LIN {X 0,Y 504.63,Z 384.162,A -85,B 0,C 180,E1 24334.794,E2 24334.794} C_VEL
LIN {X 0,Y 504.69,Z 384.156,A -85,B 0,C 180,E1 24331.534,E2 24331.534} C_VEL
LIN {X 0,Y 504.631,Z 384.188,A -85,B 0,C 180,E1 24328.264,E2 24328.264} C_VEL
LIN {X 0,Y 504.665,Z 384.158,A -85,B 0,C 180,E1 24324.835,E2 24324.835} C_VEL
LIN {X 0,Y 504.642,Z 384.183,A -85,B 0,C 180,E1 24321.624,E2 24321.624} C_VEL
LIN {X 0,Y 504.635,Z 384.173,A -85,B 0,C 180,E1 24318.123,E2 24318.123} C_VEL
LIN {X 0,Y 504.698,Z 384.163,A -85,B 0,C 180,E1 24314.806,E2 24314.806} C_VEL
LIN {X 0,Y 504.631,Z 384.169,A -85,B 0,C 180,E1 24311.428,E2 24311.428} C_VEL
LIN {X 0,Y 504.655,Z 384.173,A -85,B 0,C 180,E1 24307.972,E2 24307.972} C_VEL
LIN {X 0,Y 504.654,Z 384.182,A -85,B 0,C 180,E1 24304.773,E2 24304.773} C_VEL
LIN {X 0,Y 504.638,Z 384.181,A -85,B 0,C 180,E1 24301.362,E2 24301.362} C_VEL
LIN {X 0,Y 504.698,Z 384.182,A -85,B 0,C 180,E1 24298.07,E2 24298.07} C_VEL
LIN {X 0,Y 504.638,Z 384.185,A -85,B 0,C 180,E1 24294.656,E2 24294.656} C_VEL
LIN {X 0,Y 504.65,Z 384.184,A -85,B 0,C 180,E1 24291.11,E2 24291.11} C_VEL
LIN {X 0,Y 504.686,Z 384.178,A -85,B 0,C 180,E1 24287.761,E2 24287.761} C_VEL
LIN {X 0,Y 504.637,Z 384.18,A -85,B 0,C 180,E1 24284.485,E2 24284.485} C_VEL
LIN {X 0,Y 504.698,Z 384.175,A -85,B 0,C 180,E1 24281.16,E2 24281.16} C_VEL
LIN {X 0,Y 504.641,Z 384.178,A -85,B 0,C 180,E1 24277.886,E2 24277.886} C_VEL
LIN {X 0,Y 504.651,Z 384.179,A -85,B 0,C 180,E1 24274.355,E2 24274.355} C_VEL
LIN {X 0,Y 504.681,Z 384.161,A -85,B 0,C 180,E1 24271.092,E2 24271.092} C_VEL
LIN {X 0,Y 504.641,Z 384.182,A -85,B 0,C 180,E1 24267.659,E2 24267.659} C_VEL
LIN {X 0,Y 504.678,Z 384.151,A -85,B 0,C 180,E1 24264.236,E2 24264.236} C_VEL
LIN {X 0,Y 504.657,Z 384.186,A -85,B 0,C 180,E1 24260.946,E2 24260.946} C_VEL
LIN {X 0,Y 504.647,Z 384.176,A -85,B 0,C 180,E1 24257.481,E2 24257.481} C_VEL
LIN {X 0,Y 504.699,Z 384.152,A -85,B 0,C 180,E1 24254.148,E2 24254.148} C_VEL
LIN {X 0,Y 504.712,Z 384.421,A -85,B 0,C 180,E1 24252.343,E2 24252.343} C_VEL
LIN {X 0,Y 505.96,Z 387.581,A -85,B 0,C 180,E1 24251.839,E2 24251.839} C_VEL
LIN {X 0,Y 506.781,Z 388.94,A -85,B 0,C 180,E1 24251.616,E2 24251.616} C_VEL
LIN {X 0,Y 508.029,Z 395.982,A -85,B 0,C 180,E1 24250.823,E2 24250.823} C_VEL
LIN {X 0,Y 509.186,Z 410.16,A -85,B 0,C 180,E1 24249.409,E2 24249.409} C_VEL
LIN {X 0,Y 510.462,Z 414.617,A -85,B 0,C 180,E1 24248.871,E2 24248.871} C_VEL
LIN {X 0,Y 513.393,Z 421.793,A -85,B 0,C 180,E1 24247.93,E2 24247.93} C_VEL
LIN {X 0,Y 510.149,Z 468.492,A -85,B 0,C 180,E1 24244.297,E2 24244.297} C_VEL
LIN {X 0,Y 510.416,Z 471.577,A -85,B 0,C 180,E1 24244.143,E2 24244.143} C_VEL
LIN {X 0,Y 513.342,Z 489.328,A -85,B 0,C 180,E1 24243.576,E2 24243.576} C_VEL
LIN {X 0,Y 510.537,Z 702.166,A -85,B 0,C 180,E1 24240.34,E2 24240.34} C_VEL
LIN {X 0,Y 509.946,Z 737.203,A -85,B 0,C 180,E1 24239.76,E2 24239.76} C_VEL
LIN {X 0,Y 509.167,Z 757.239,A -85,B 0,C 180,E1 24239.22,E2 24239.22} C_VEL
LIN {X 0,Y 508.146,Z 775.437,A -85,B 0,C 180,E1 24238.532,E2 24238.532} C_VEL
LIN {X 0,Y 506.819,Z 794.151,A -85,B 0,C 180,E1 24237.621,E2 24237.621} C_VEL
LIN {X 0,Y 505.413,Z 811.582,A -85,B 0,C 180,E1 24236.558,E2 24236.558} C_VEL
LIN {X 0,Y 503.7,Z 829.704,A -85,B 0,C 180,E1 24235.201,E2 24235.201} C_VEL
LIN {X 0,Y 502.073,Z 846.017,A -85,B 0,C 180,E1 24233.721,E2 24233.721} C_VEL
LIN {X 0,Y 500.46,Z 861.756,A -85,B 0,C 180,E1 24232.025,E2 24232.025} C_VEL
LIN {X 0,Y 498.795,Z 880.019,A -85,B 0,C 180,E1 24229.68,E2 24229.68} C_VEL
LIN {X 0,Y 497.903,Z 893.059,A -85,B 0,C 180,E1 24227.773,E2 24227.773} C_VEL
LIN {X 0,Y 497.196,Z 904.769,A -85,B 0,C 180,E1 24225.753,E2 24225.753} C_VEL
LIN {X 0,Y 496.636,Z 915.718,A -85,B 0,C 180,E1 24223.49,E2 24223.49} C_VEL
LIN {X 0,Y 496.275,Z 924.505,A -85,B 0,C 180,E1 24221.27,E2 24221.27} C_VEL
LIN {X 0,Y 496.064,Z 931.644,A -85,B 0,C 180,E1 24219.018,E2 24219.018} C_VEL
LIN {X 0,Y 495.966,Z 937.163,A -85,B 0,C 180,E1 24216.715,E2 24216.715} C_VEL
LIN {X 0,Y 495.923,Z 941.025,A -85,B 0,C 180,E1 24214.394,E2 24214.394} C_VEL
LIN {X 0,Y 495.913,Z 943.345,A -85,B 0,C 180,E1 24211.964,E2 24211.964} C_VEL
LIN {X 0,Y 495.903,Z 943.948,A -85,B 0,C 180,E1 24209.653,E2 24209.653} C_VEL
LIN {X 0,Y 495.907,Z 942.989,A -85,B 0,C 180,E1 24207.342,E2 24207.342} C_VEL
LIN {X 0,Y 495.924,Z 940.351,A -85,B 0,C 180,E1 24205.026,E2 24205.026} C_VEL
LIN {X 0,Y 495.968,Z 936.05,A -85,B 0,C 180,E1 24202.686,E2 24202.686} C_VEL
LIN {X 0,Y 496.099,Z 930.109,A -85,B 0,C 180,E1 24200.37,E2 24200.37} C_VEL
LIN {X 0,Y 496.343,Z 922.728,A -85,B 0,C 180,E1 24198.143,E2 24198.143} C_VEL
LIN {X 0,Y 496.74,Z 913.462,A -85,B 0,C 180,E1 24195.904,E2 24195.904} C_VEL
LIN {X 0,Y 497.314,Z 902.703,A -85,B 0,C 180,E1 24193.772,E2 24193.772} C_VEL
LIN {X 0,Y 498.082,Z 890.332,A -85,B 0,C 180,E1 24191.716,E2 24191.716} C_VEL
LIN {X 0,Y 499.412,Z 872.531,A -85,B 0,C 180,E1 24189.224,E2 24189.224} C_VEL
LIN {X 0,Y 500.948,Z 857.086,A -85,B 0,C 180,E1 24187.343,E2 24187.343} C_VEL
LIN {X 0,Y 502.625,Z 840.515,A -85,B 0,C 180,E1 24185.657,E2 24185.657} C_VEL
LIN {X 0,Y 504.236,Z 824.047,A -85,B 0,C 180,E1 24184.262,E2 24184.262} C_VEL
LIN {X 0,Y 505.82,Z 806.472,A -85,B 0,C 180,E1 24183.021,E2 24183.021} C_VEL
LIN {X 0,Y 507.308,Z 787.941,A -85,B 0,C 180,E1 24181.961,E2 24181.961} C_VEL
LIN {X 0,Y 508.538,Z 769.216,A -85,B 0,C 180,E1 24181.114,E2 24181.114} C_VEL
LIN {X 0,Y 509.525,Z 749.435,A -85,B 0,C 180,E1 24180.455,E2 24180.455} C_VEL
LIN {X 0,Y 510.109,Z 729.43,A -85,B 0,C 180,E1 24179.999,E2 24179.999} C_VEL
LIN {X 0,Y 512.344,Z 567.172,A -85,B 0,C 180,E1 24177.509,E2 24177.509} C_VEL
LIN {X 0,Y 513.183,Z 487.495,A -85,B 0,C 180,E1 24176.288,E2 24176.288} C_VEL
LIN {X 0,Y 510.105,Z 469.195,A -85,B 0,C 180,E1 24175.665,E2 24175.665} C_VEL
LIN {X 0,Y 513.299,Z 423.111,A -85,B 0,C 180,E1 24172.083,E2 24172.083} C_VEL
LIN {X 0,Y 513.288,Z 421.061,A -85,B 0,C 180,E1 24171.904,E2 24171.904} C_VEL
LIN {X 0,Y 506.083,Z 405.037,A -85,B 0,C 180,E1 24169.695,E2 24169.695} C_VEL
LIN {X 0,Y 499.801,Z 392.121,A -85,B 0,C 180,E1 24167.748,E2 24167.748} C_VEL
LIN {X 0,Y 498.273,Z 389.006,A -85,B 0,C 180,E1 24167.26,E2 24167.26} C_VEL
LIN {X 0,Y 496.757,Z 385.456,A -85,B 0,C 180,E1 24166.679,E2 24166.679} C_VEL
LIN {X 0,Y 496.718,Z 385.143,A -85,B 0,C 180,E1 24165.208,E2 24165.208} C_VEL
LIN {X 0,Y 496.764,Z 385.142,A -85,B 0,C 180,E1 24161.776,E2 24161.776} C_VEL
LIN {X 0,Y 496.711,Z 385.175,A -85,B 0,C 180,E1 24158.46,E2 24158.46} C_VEL
LIN {X 0,Y 496.732,Z 385.147,A -85,B 0,C 180,E1 24154.991,E2 24154.991} C_VEL
LIN {X 0,Y 496.738,Z 385.152,A -85,B 0,C 180,E1 24151.631,E2 24151.631} C_VEL
LIN {X 0,Y 496.708,Z 385.17,A -85,B 0,C 180,E1 24148.153,E2 24148.153} C_VEL
LIN {X 0,Y 496.752,Z 385.166,A -85,B 0,C 180,E1 24144.75,E2 24144.75} C_VEL
LIN {X 0,Y 496.721,Z 385.165,A -85,B 0,C 180,E1 24141.367,E2 24141.367} C_VEL
LIN {X 0,Y 496.705,Z 385.172,A -85,B 0,C 180,E1 24137.817,E2 24137.817} C_VEL
LIN {X 0,Y 496.769,Z 385.161,A -85,B 0,C 180,E1 24134.453,E2 24134.453} C_VEL
LIN {X 0,Y 496.711,Z 385.162,A -85,B 0,C 180,E1 24131.025,E2 24131.025} C_VEL
LIN {X 0,Y 496.706,Z 385.164,A -85,B 0,C 180,E1 24127.519,E2 24127.519} C_VEL
LIN {X 0,Y 496.76,Z 385.164,A -85,B 0,C 180,E1 24124.156,E2 24124.156} C_VEL
LIN {X 0,Y 496.7,Z 385.172,A -85,B 0,C 180,E1 24120.808,E2 24120.808} C_VEL
LIN {X 0,Y 496.723,Z 385.171,A -85,B 0,C 180,E1 24117.347,E2 24117.347} C_VEL
LIN {X 0,Y 496.732,Z 385.172,A -85,B 0,C 180,E1 24113.992,E2 24113.992} C_VEL
LIN {X 0,Y 496.697,Z 385.174,A -85,B 0,C 180,E1 24110.535,E2 24110.535} C_VEL
LIN {X 0,Y 496.737,Z 385.132,A -85,B 0,C 180,E1 24107.09,E2 24107.09} C_VEL
LIN {X 0,Y 496.704,Z 385.172,A -85,B 0,C 180,E1 24103.872,E2 24103.872} C_VEL
LIN {X 0,Y 496.698,Z 385.138,A -85,B 0,C 180,E1 24100.357,E2 24100.357} C_VEL
LIN {X 0,Y 496.758,Z 385.17,A -85,B 0,C 180,E1 24097.016,E2 24097.016} C_VEL
LIN {X 0,Y 496.693,Z 385.151,A -85,B 0,C 180,E1 24093.585,E2 24093.585} C_VEL
LIN {X 0,Y 496.704,Z 385.148,A -85,B 0,C 180,E1 24090.052,E2 24090.052} C_VEL
LIN {X 0,Y 496.728,Z 385.177,A -85,B 0,C 180,E1 24086.804,E2 24086.804} C_VEL
LIN {X 0,Y 496.689,Z 385.16,A -85,B 0,C 180,E1 24083.426,E2 24083.426} C_VEL
LIN {X 0,Y 496.775,Z 385.4,A -85,B 0,C 180,E1 24082.468,E2 24082.468} C_VEL
LIN {X 0,Y 497.335,Z 387.314,A -85,B 0,C 180,E1 24082.181,E2 24082.181} C_VEL
LIN {X 0,Y 499.538,Z 390.989,A -85,B 0,C 180,E1 24081.649,E2 24081.649} C_VEL
LIN {X 0,Y 507.023,Z 404.592,A -85,B 0,C 180,E1 24079.846,E2 24079.846} C_VEL
LIN {X 0,Y 517.059,Z 423.783,A -85,B 0,C 180,E1 24077.556,E2 24077.556} C_VEL
LIN {X 0,Y 519.732,Z 428.932,A -85,B 0,C 180,E1 24076.974,E2 24076.974} C_VEL
LIN {X 0,Y 518.222,Z 466.463,A -85,B 0,C 180,E1 24074.906,E2 24074.906} C_VEL
LIN {X 0,Y 520.792,Z 487.007,A -85,B 0,C 180,E1 24074.305,E2 24074.305} C_VEL
LIN {X 0,Y 518.435,Z 664.252,A -85,B 0,C 180,E1 24071.478,E2 24071.478} C_VEL
LIN {X 0,Y 516.725,Z 807.877,A -85,B 0,C 180,E1 24069.261,E2 24069.261} C_VEL
LIN {X 0,Y 515.915,Z 829.827,A -85,B 0,C 180,E1 24068.805,E2 24068.805} C_VEL
LIN {X 0,Y 514.717,Z 853.373,A -85,B 0,C 180,E1 24068.099,E2 24068.099} C_VEL
LIN {X 0,Y 513.479,Z 872.878,A -85,B 0,C 180,E1 24067.342,E2 24067.342} C_VEL
LIN {X 0,Y 511.818,Z 894.667,A -85,B 0,C 180,E1 24066.294,E2 24066.294} C_VEL
LIN {X 0,Y 510.105,Z 914.827,A -85,B 0,C 180,E1 24065.12,E2 24065.12} C_VEL
LIN {X 0,Y 508.148,Z 936.137,A -85,B 0,C 180,E1 24063.635,E2 24063.635} C_VEL
LIN {X 0,Y 506.3,Z 955.179,A -85,B 0,C 180,E1 24062.089,E2 24062.089} C_VEL
LIN {X 0,Y 504.41,Z 973.998,A -85,B 0,C 180,E1 24060.297,E2 24060.297} C_VEL
LIN {X 0,Y 502.616,Z 992.054,A -85,B 0,C 180,E1 24058.324,E2 24058.324} C_VEL
LIN {X 0,Y 501.065,Z 1008.11,A -85,B 0,C 180,E1 24056.295,E2 24056.295} C_VEL
LIN {X 0,Y 499.605,Z 1024.117,A -85,B 0,C 180,E1 24053.971,E2 24053.971} C_VEL
LIN {X 0,Y 498.468,Z 1037.954,A -85,B 0,C 180,E1 24051.659,E2 24051.659} C_VEL
LIN {X 0,Y 497.559,Z 1050.297,A -85,B 0,C 180,E1 24049.242,E2 24049.242} C_VEL
LIN {X 0,Y 496.88,Z 1061.479,A -85,B 0,C 180,E1 24046.698,E2 24046.698} C_VEL
LIN {X 0,Y 496.45,Z 1070.152,A -85,B 0,C 180,E1 24044.343,E2 24044.343} C_VEL
LIN {X 0,Y 496.149,Z 1078.436,A -85,B 0,C 180,E1 24041.626,E2 24041.626} C_VEL
LIN {X 0,Y 496.008,Z 1084.082,A -85,B 0,C 180,E1 24039.28,E2 24039.28} C_VEL
LIN {X 0,Y 495.933,Z 1089.001,A -85,B 0,C 180,E1 24036.599,E2 24036.599} C_VEL
LIN {X 0,Y 495.915,Z 1091.956,A -85,B 0,C 180,E1 24034.162,E2 24034.162} C_VEL
LIN {X 0,Y 495.909,Z 1093.714,A -85,B 0,C 180,E1 24031.502,E2 24031.502} C_VEL
LIN {X 0,Y 495.89,Z 1093.827,A -85,B 0,C 180,E1 24029.076,E2 24029.076} C_VEL
LIN {X 0,Y 495.89,Z 1092.631,A -85,B 0,C 180,E1 24026.532,E2 24026.532} C_VEL
LIN {X 0,Y 495.916,Z 1089.799,A -85,B 0,C 180,E1 24023.982,E2 24023.982} C_VEL
LIN {X 0,Y 495.991,Z 1085.598,A -85,B 0,C 180,E1 24021.421,E2 24021.421} C_VEL
LIN {X 0,Y 496.106,Z 1079.653,A -85,B 0,C 180,E1 24018.844,E2 24018.844} C_VEL
LIN {X 0,Y 496.365,Z 1072.176,A -85,B 0,C 180,E1 24016.249,E2 24016.249} C_VEL
LIN {X 0,Y 496.78,Z 1063.212,A -85,B 0,C 180,E1 24013.748,E2 24013.748} C_VEL
LIN {X 0,Y 497.442,Z 1052.019,A -85,B 0,C 180,E1 24011.118,E2 24011.118} C_VEL
LIN {X 0,Y 498.267,Z 1040.541,A -85,B 0,C 180,E1 24008.826,E2 24008.826} C_VEL
LIN {X 0,Y 499.407,Z 1026.428,A -85,B 0,C 180,E1 24006.395,E2 24006.395} C_VEL
LIN {X 0,Y 500.727,Z 1011.743,A -85,B 0,C 180,E1 24004.195,E2 24004.195} C_VEL
LIN {X 0,Y 502.264,Z 995.601,A -85,B 0,C 180,E1 24002.107,E2 24002.107} C_VEL
LIN {X 0,Y 504.038,Z 977.863,A -85,B 0,C 180,E1 24000.097,E2 24000.097} C_VEL
LIN {X 0,Y 505.815,Z 959.917,A -85,B 0,C 180,E1 23998.343,E2 23998.343} C_VEL
LIN {X 0,Y 507.86,Z 939.085,A -85,B 0,C 180,E1 23996.59,E2 23996.59} C_VEL
LIN {X 0,Y 509.706,Z 919.625,A -85,B 0,C 180,E1 23995.191,E2 23995.191} C_VEL
LIN {X 0,Y 511.52,Z 898.059,A -85,B 0,C 180,E1 23993.89,E2 23993.89} C_VEL
LIN {X 0,Y 513.284,Z 875.978,A -85,B 0,C 180,E1 23992.789,E2 23992.789} C_VEL
LIN {X 0,Y 514.633,Z 854.816,A -85,B 0,C 180,E1 23991.952,E2 23991.952} C_VEL
LIN {X 0,Y 515.817,Z 832.781,A -85,B 0,C 180,E1 23991.268,E2 23991.268} C_VEL
LIN {X 0,Y 516.657,Z 810.082,A -85,B 0,C 180,E1 23990.779,E2 23990.779} C_VEL
LIN {X 0,Y 517.852,Z 716.781,A -85,B 0,C 180,E1 23989.33,E2 23989.33} C_VEL
LIN {X 0,Y 519.994,Z 539.646,A -85,B 0,C 180,E1 23986.553,E2 23986.553} C_VEL
LIN {X 0,Y 520.642,Z 484.455,A -85,B 0,C 180,E1 23985.636,E2 23985.636} C_VEL
LIN {X 0,Y 518.15,Z 464.866,A -85,B 0,C 180,E1 23985.029,E2 23985.029} C_VEL
LIN {X 0,Y 519.727,Z 428.905,A -85,B 0,C 180,E1 23983.025,E2 23983.025} C_VEL
LIN {X 0,Y 508.024,Z 406.493,A -85,B 0,C 180,E1 23980.388,E2 23980.388} C_VEL
LIN {X 0,Y 501.28,Z 394.127,A -85,B 0,C 180,E1 23978.778,E2 23978.778} C_VEL
LIN {X 0,Y 498.664,Z 389.47,A -85,B 0,C 180,E1 23978.138,E2 23978.138} C_VEL
LIN {X 0,Y 496.911,Z 386.03,A -85,B 0,C 180,E1 23977.671,E2 23977.671} C_VEL
LIN {X 0,Y 496.735,Z 385.187,A -85,B 0,C 180,E1 23977.436,E2 23977.436} C_VEL
LIN {X 0,Y 496.7,Z 385.157,A -85,B 0,C 180,E1 23974.168,E2 23974.168} C_VEL
LIN {X 0,Y 496.689,Z 385.144,A -85,B 0,C 180,E1 23970.617,E2 23970.617} C_VEL
LIN {X 0,Y 496.754,Z 385.161,A -85,B 0,C 180,E1 23967.317,E2 23967.317} C_VEL
LIN {X 0,Y 496.696,Z 385.166,A -85,B 0,C 180,E1 23963.867,E2 23963.867} C_VEL
LIN {X 0,Y 496.696,Z 385.143,A -85,B 0,C 180,E1 23960.257,E2 23960.257} C_VEL
LIN {X 0,Y 496.759,Z 385.168,A -85,B 0,C 180,E1 23956.848,E2 23956.848} C_VEL
LIN {X 0,Y 496.69,Z 385.14,A -85,B 0,C 180,E1 23953.504,E2 23953.504} C_VEL
LIN {X 0,Y 496.712,Z 385.171,A -85,B 0,C 180,E1 23949.969,E2 23949.969} C_VEL
LIN {X 0,Y 496.73,Z 385.165,A -85,B 0,C 180,E1 23946.704,E2 23946.704} C_VEL
LIN {X 0,Y 496.694,Z 385.169,A -85,B 0,C 180,E1 23943.231,E2 23943.231} C_VEL
LIN {X 0,Y 496.735,Z 385.167,A -85,B 0,C 180,E1 23939.769,E2 23939.769} C_VEL
LIN {X 0,Y 496.715,Z 385.166,A -85,B 0,C 180,E1 23936.422,E2 23936.422} C_VEL
LIN {X 0,Y 496.698,Z 385.165,A -85,B 0,C 180,E1 23932.942,E2 23932.942} C_VEL
LIN {X 0,Y 496.759,Z 385.162,A -85,B 0,C 180,E1 23929.563,E2 23929.563} C_VEL
LIN {X 0,Y 496.702,Z 385.174,A -85,B 0,C 180,E1 23926.259,E2 23926.259} C_VEL
LIN {X 0,Y 496.709,Z 385.171,A -85,B 0,C 180,E1 23922.667,E2 23922.667} C_VEL
LIN {X 0,Y 496.765,Z 385.169,A -85,B 0,C 180,E1 23919.253,E2 23919.253} C_VEL
LIN {X 0,Y 496.702,Z 385.175,A -85,B 0,C 180,E1 23915.88,E2 23915.88} C_VEL
LIN {X 0,Y 496.719,Z 385.17,A -85,B 0,C 180,E1 23912.337,E2 23912.337} C_VEL
LIN {X 0,Y 496.743,Z 385.137,A -85,B 0,C 180,E1 23908.983,E2 23908.983} C_VEL
LIN {X 0,Y 496.702,Z 385.165,A -85,B 0,C 180,E1 23905.552,E2 23905.552} C_VEL
LIN {X 0,Y 496.738,Z 385.166,A -85,B 0,C 180,E1 23902.096,E2 23902.096} C_VEL
LIN {X 0,Y 496.717,Z 385.142,A -85,B 0,C 180,E1 23898.835,E2 23898.835} C_VEL
LIN {X 0,Y 496.706,Z 385.152,A -85,B 0,C 180,E1 23895.369,E2 23895.369} C_VEL
LIN {X 0,Y 496.732,Z 385.35,A -85,B 0,C 180,E1 23893.265,E2 23893.265} C_VEL
LIN {X 0,Y 497.231,Z 387.193,A -85,B 0,C 180,E1 23892.949,E2 23892.949} C_VEL
LIN {X 0,Y 499.228,Z 390.844,A -85,B 0,C 180,E1 23892.35,E2 23892.35} C_VEL
LIN {X 0,Y 506.688,Z 406.327,A -85,B 0,C 180,E1 23890.035,E2 23890.035} C_VEL
LIN {X 0,Y 510.462,Z 414.617,A -85,B 0,C 180,E1 23888.871,E2 23888.871} C_VEL
LIN {X 0,Y 510.841,Z 417.844,A -85,B 0,C 180,E1 23888.545,E2 23888.545} C_VEL
LIN {X 0,Y 509.505,Z 423.566,A -85,B 0,C 180,E1 23888.182,E2 23888.182} C_VEL
LIN {X 0,Y 506.401,Z 433.052,A -85,B 0,C 180,E1 23887.673,E2 23887.673} C_VEL
LIN {X 0,Y 506.114,Z 435.006,A -85,B 0,C 180,E1 23887.531,E2 23887.531} C_VEL
LIN {X 0,Y 503.717,Z 470.182,A -85,B 0,C 180,E1 23884.808,E2 23884.808} C_VEL
LIN {X 0,Y 507.166,Z 490.554,A -85,B 0,C 180,E1 23884.134,E2 23884.134} C_VEL
LIN {X 0,Y 504.221,Z 712.5,A -85,B 0,C 180,E1 23880.761,E2 23880.761} C_VEL
LIN {X 0,Y 503.713,Z 739.739,A -85,B 0,C 180,E1 23880.289,E2 23880.289} C_VEL
LIN {X 0,Y 502.928,Z 759.685,A -85,B 0,C 180,E1 23879.738,E2 23879.738} C_VEL
LIN {X 0,Y 501.799,Z 778.126,A -85,B 0,C 180,E1 23879.018,E2 23879.018} C_VEL
LIN {X 0,Y 500.345,Z 796.898,A -85,B 0,C 180,E1 23878.074,E2 23878.074} C_VEL
LIN {X 0,Y 498.733,Z 814.822,A -85,B 0,C 180,E1 23876.942,E2 23876.942} C_VEL
LIN {X 0,Y 496.983,Z 831.91,A -85,B 0,C 180,E1 23875.63,E2 23875.63} C_VEL
LIN {X 0,Y 495.142,Z 848.623,A -85,B 0,C 180,E1 23874.074,E2 23874.074} C_VEL
LIN {X 0,Y 493.347,Z 864.276,A -85,B 0,C 180,E1 23872.334,E2 23872.334} C_VEL
LIN {X 0,Y 491.786,Z 878.408,A -85,B 0,C 180,E1 23870.469,E2 23870.469} C_VEL
LIN {X 0,Y 490.405,Z 891.541,A -85,B 0,C 180,E1 23868.423,E2 23868.423} C_VEL
LIN {X 0,Y 489.111,Z 908.478,A -85,B 0,C 180,E1 23865.29,E2 23865.29} C_VEL
LIN {X 0,Y 488.576,Z 918.71,A -85,B 0,C 180,E1 23863.01,E2 23863.01} C_VEL
LIN {X 0,Y 488.218,Z 927.339,A -85,B 0,C 180,E1 23860.621,E2 23860.621} C_VEL
LIN {X 0,Y 488.026,Z 933.998,A -85,B 0,C 180,E1 23858.246,E2 23858.246} C_VEL
LIN {X 0,Y 487.944,Z 938.888,A -85,B 0,C 180,E1 23855.881,E2 23855.881} C_VEL
LIN {X 0,Y 487.905,Z 942.234,A -85,B 0,C 180,E1 23853.407,E2 23853.407} C_VEL
LIN {X 0,Y 487.908,Z 943.794,A -85,B 0,C 180,E1 23851.057,E2 23851.057} C_VEL
LIN {X 0,Y 487.902,Z 943.766,A -85,B 0,C 180,E1 23848.708,E2 23848.708} C_VEL
LIN {X 0,Y 487.908,Z 942.095,A -85,B 0,C 180,E1 23846.358,E2 23846.358} C_VEL
LIN {X 0,Y 487.947,Z 938.837,A -85,B 0,C 180,E1 23844.001,E2 23844.001} C_VEL
LIN {X 0,Y 488.032,Z 933.924,A -85,B 0,C 180,E1 23841.636,E2 23841.636} C_VEL
LIN {X 0,Y 488.221,Z 927.242,A -85,B 0,C 180,E1 23839.259,E2 23839.259} C_VEL
LIN {X 0,Y 488.584,Z 918.589,A -85,B 0,C 180,E1 23836.87,E2 23836.87} C_VEL
LIN {X 0,Y 489.122,Z 908.328,A -85,B 0,C 180,E1 23834.589,E2 23834.589} C_VEL
LIN {X 0,Y 490.428,Z 891.298,A -85,B 0,C 180,E1 23831.445,E2 23831.445} C_VEL
LIN {X 0,Y 491.814,Z 878.172,A -85,B 0,C 180,E1 23829.408,E2 23829.408} C_VEL
LIN {X 0,Y 493.386,Z 863.912,A -85,B 0,C 180,E1 23827.533,E2 23827.533} C_VEL
LIN {X 0,Y 495.07,Z 849.336,A -85,B 0,C 180,E1 23825.906,E2 23825.906} C_VEL
LIN {X 0,Y 496.881,Z 832.785,A -85,B 0,C 180,E1 23824.356,E2 23824.356} C_VEL
LIN {X 0,Y 498.612,Z 815.988,A -85,B 0,C 180,E1 23823.051,E2 23823.051} C_VEL
LIN {X 0,Y 500.317,Z 797.317,A -85,B 0,C 180,E1 23821.859,E2 23821.859} C_VEL
LIN {X 0,Y 501.778,Z 778.53,A -85,B 0,C 180,E1 23820.908,E2 23820.908} C_VEL
LIN {X 0,Y 502.93,Z 759.699,A -85,B 0,C 180,E1 23820.172,E2 23820.172} C_VEL
LIN {X 0,Y 503.724,Z 739.594,A -85,B 0,C 180,E1 23819.616,E2 23819.616} C_VEL
LIN {X 0,Y 504.304,Z 708.91,A -85,B 0,C 180,E1 23819.09,E2 23819.09} C_VEL
LIN {X 0,Y 507.145,Z 489.903,A -85,B 0,C 180,E1 23815.763,E2 23815.763} C_VEL
LIN {X 0,Y 503.646,Z 469.309,A -85,B 0,C 180,E1 23815.058,E2 23815.058} C_VEL
LIN {X 0,Y 506.849,Z 425.935,A -85,B 0,C 180,E1 23811.653,E2 23811.653} C_VEL
LIN {X 0,Y 506.593,Z 424.484,A -85,B 0,C 180,E1 23811.497,E2 23811.497} C_VEL
LIN {X 0,Y 498.873,Z 407.129,A -85,B 0,C 180,E1 23809.051,E2 23809.051} C_VEL
LIN {X 0,Y 492.732,Z 394.612,A -85,B 0,C 180,E1 23807.101,E2 23807.101} C_VEL
LIN {X 0,Y 490.44,Z 390.091,A -85,B 0,C 180,E1 23806.364,E2 23806.364} C_VEL
LIN {X 0,Y 488.87,Z 386.456,A -85,B 0,C 180,E1 23805.75,E2 23805.75} C_VEL
LIN {X 0,Y 488.771,Z 386.133,A -85,B 0,C 180,E1 23804.891,E2 23804.891} C_VEL
LIN {X 0,Y 488.821,Z 386.126,A -85,B 0,C 180,E1 23801.508,E2 23801.508} C_VEL
LIN {X 0,Y 488.783,Z 386.164,A -85,B 0,C 180,E1 23798.154,E2 23798.154} C_VEL
LIN {X 0,Y 488.773,Z 386.142,A -85,B 0,C 180,E1 23794.659,E2 23794.659} C_VEL
LIN {X 0,Y 488.828,Z 386.126,A -85,B 0,C 180,E1 23791.241,E2 23791.241} C_VEL
LIN {X 0,Y 488.774,Z 386.158,A -85,B 0,C 180,E1 23787.802,E2 23787.802} C_VEL
LIN {X 0,Y 488.772,Z 386.163,A -85,B 0,C 180,E1 23784.151,E2 23784.151} C_VEL
LIN {X 0,Y 488.828,Z 386.156,A -85,B 0,C 180,E1 23780.724,E2 23780.724} C_VEL
LIN {X 0,Y 488.777,Z 386.159,A -85,B 0,C 180,E1 23777.255,E2 23777.255} C_VEL
LIN {X 0,Y 488.767,Z 386.162,A -85,B 0,C 180,E1 23773.662,E2 23773.662} C_VEL
LIN {X 0,Y 488.821,Z 386.152,A -85,B 0,C 180,E1 23770.251,E2 23770.251} C_VEL
LIN {X 0,Y 488.767,Z 386.153,A -85,B 0,C 180,E1 23766.933,E2 23766.933} C_VEL
LIN {X 0,Y 488.766,Z 386.155,A -85,B 0,C 180,E1 23763.284,E2 23763.284} C_VEL
LIN {X 0,Y 488.831,Z 386.148,A -85,B 0,C 180,E1 23759.883,E2 23759.883} C_VEL
LIN {X 0,Y 488.771,Z 386.157,A -85,B 0,C 180,E1 23756.365,E2 23756.365} C_VEL
LIN {X 0,Y 488.762,Z 386.155,A -85,B 0,C 180,E1 23752.826,E2 23752.826} C_VEL
LIN {X 0,Y 488.818,Z 386.149,A -85,B 0,C 180,E1 23749.392,E2 23749.392} C_VEL
LIN {X 0,Y 488.766,Z 386.132,A -85,B 0,C 180,E1 23745.911,E2 23745.911} C_VEL
LIN {X 0,Y 488.76,Z 386.154,A -85,B 0,C 180,E1 23742.377,E2 23742.377} C_VEL
LIN {X 0,Y 488.818,Z 386.136,A -85,B 0,C 180,E1 23738.9,E2 23738.9} C_VEL
LIN {X 0,Y 488.759,Z 386.14,A -85,B 0,C 180,E1 23735.553,E2 23735.553} C_VEL
LIN {X 0,Y 488.759,Z 386.166,A -85,B 0,C 180,E1 23731.933,E2 23731.933} C_VEL
LIN {X 0,Y 488.817,Z 386.127,A -85,B 0,C 180,E1 23728.536,E2 23728.536} C_VEL
LIN {X 0,Y 488.755,Z 386.134,A -85,B 0,C 180,E1 23725.119,E2 23725.119} C_VEL
LIN {X 0,Y 488.777,Z 386.339,A -85,B 0,C 180,E1 23723.468,E2 23723.468} C_VEL
LIN {X 0,Y 489.126,Z 387.771,A -85,B 0,C 180,E1 23723.206,E2 23723.206} C_VEL
LIN {X 0,Y 490.839,Z 390.609,A -85,B 0,C 180,E1 23722.772,E2 23722.772} C_VEL
LIN {X 0,Y 491.719,Z 392.028,A -85,B 0,C 180,E1 23722.557,E2 23722.557} C_VEL
LIN {X 0,Y 499.913,Z 406.983,A -85,B 0,C 180,E1 23720.505,E2 23720.505} C_VEL
LIN {X 0,Y 508.002,Z 422.231,A -85,B 0,C 180,E1 23718.6,E2 23718.6} C_VEL
LIN {X 0,Y 513.383,Z 432.894,A -85,B 0,C 180,E1 23717.37,E2 23717.37} C_VEL
LIN {X 0,Y 511.861,Z 466.596,A -85,B 0,C 180,E1 23715.487,E2 23715.487} C_VEL
LIN {X 0,Y 514.518,Z 488.474,A -85,B 0,C 180,E1 23714.838,E2 23714.838} C_VEL
LIN {X 0,Y 511.682,Z 670.904,A -85,B 0,C 180,E1 23711.868,E2 23711.868} C_VEL
LIN {X 0,Y 509.777,Z 816.978,A -85,B 0,C 180,E1 23709.587,E2 23709.587} C_VEL
LIN {X 0,Y 508.897,Z 840.153,A -85,B 0,C 180,E1 23709.042,E2 23709.042} C_VEL
LIN {X 0,Y 507.956,Z 859.364,A -85,B 0,C 180,E1 23708.437,E2 23708.437} C_VEL
LIN {X 0,Y 506.388,Z 881.086,A -85,B 0,C 180,E1 23707.527,E2 23707.527} C_VEL
LIN {X 0,Y 504.635,Z 901.843,A -85,B 0,C 180,E1 23706.446,E2 23706.446} C_VEL
LIN {X 0,Y 502.734,Z 922.062,A -85,B 0,C 180,E1 23705.174,E2 23705.174} C_VEL
LIN {X 0,Y 500.808,Z 941.004,A -85,B 0,C 180,E1 23703.781,E2 23703.781} C_VEL
LIN {X 0,Y 498.698,Z 960.588,A -85,B 0,C 180,E1 23702.094,E2 23702.094} C_VEL
LIN {X 0,Y 496.762,Z 978.721,A -85,B 0,C 180,E1 23700.292,E2 23700.292} C_VEL
LIN {X 0,Y 494.906,Z 995.601,A -85,B 0,C 180,E1 23698.345,E2 23698.345} C_VEL
LIN {X 0,Y 493.238,Z 1011.744,A -85,B 0,C 180,E1 23696.226,E2 23696.226} C_VEL
LIN {X 0,Y 491.782,Z 1026.427,A -85,B 0,C 180,E1 23693.993,E2 23693.993} C_VEL
LIN {X 0,Y 490.518,Z 1040.542,A -85,B 0,C 180,E1 23691.525,E2 23691.525} C_VEL
LIN {X 0,Y 489.62,Z 1052.014,A -85,B 0,C 180,E1 23689.195,E2 23689.195} C_VEL
LIN {X 0,Y 488.91,Z 1062.772,A -85,B 0,C 180,E1 23686.637,E2 23686.637} C_VEL
LIN {X 0,Y 488.456,Z 1071.367,A -85,B 0,C 180,E1 23684.22,E2 23684.22} C_VEL
LIN {X 0,Y 488.154,Z 1079.046,A -85,B 0,C 180,E1 23681.58,E2 23681.58} C_VEL
LIN {X 0,Y 488.015,Z 1084.591,A -85,B 0,C 180,E1 23679.196,E2 23679.196} C_VEL
LIN {X 0,Y 487.939,Z 1089.459,A -85,B 0,C 180,E1 23676.369,E2 23676.369} C_VEL
LIN {X 0,Y 487.914,Z 1092.182,A -85,B 0,C 180,E1 23673.995,E2 23673.995} C_VEL
LIN {X 0,Y 487.908,Z 1093.759,A -85,B 0,C 180,E1 23671.292,E2 23671.292} C_VEL
LIN {X 0,Y 487.896,Z 1093.804,A -85,B 0,C 180,E1 23668.943,E2 23668.943} C_VEL
LIN {X 0,Y 487.905,Z 1092.407,A -85,B 0,C 180,E1 23666.24,E2 23666.24} C_VEL
LIN {X 0,Y 487.931,Z 1089.639,A -85,B 0,C 180,E1 23663.765,E2 23663.765} C_VEL
LIN {X 0,Y 488.007,Z 1085.099,A -85,B 0,C 180,E1 23661.042,E2 23661.042} C_VEL
LIN {X 0,Y 488.14,Z 1079.349,A -85,B 0,C 180,E1 23658.54,E2 23658.54} C_VEL
LIN {X 0,Y 488.438,Z 1071.771,A -85,B 0,C 180,E1 23655.901,E2 23655.901} C_VEL
LIN {X 0,Y 488.88,Z 1063.234,A -85,B 0,C 180,E1 23653.484,E2 23653.484} C_VEL
LIN {X 0,Y 489.58,Z 1052.591,A -85,B 0,C 180,E1 23650.927,E2 23650.927} C_VEL
LIN {X 0,Y 490.467,Z 1041.18,A -85,B 0,C 180,E1 23648.598,E2 23648.598} C_VEL
LIN {X 0,Y 491.782,Z 1026.426,A -85,B 0,C 180,E1 23646.007,E2 23646.007} C_VEL
LIN {X 0,Y 493.238,Z 1011.744,A -85,B 0,C 180,E1 23643.774,E2 23643.774} C_VEL
LIN {X 0,Y 494.905,Z 995.6,A -85,B 0,C 180,E1 23641.655,E2 23641.655} C_VEL
LIN {X 0,Y 496.81,Z 978.245,A -85,B 0,C 180,E1 23639.658,E2 23639.658} C_VEL
LIN {X 0,Y 498.768,Z 959.914,A -85,B 0,C 180,E1 23637.843,E2 23637.843} C_VEL
LIN {X 0,Y 500.97,Z 939.375,A -85,B 0,C 180,E1 23636.093,E2 23636.093} C_VEL
LIN {X 0,Y 502.888,Z 920.522,A -85,B 0,C 180,E1 23634.719,E2 23634.719} C_VEL
LIN {X 0,Y 504.852,Z 899.186,A -85,B 0,C 180,E1 23633.406,E2 23633.406} C_VEL
LIN {X 0,Y 506.639,Z 878.388,A -85,B 0,C 180,E1 23632.345,E2 23632.345} C_VEL
LIN {X 0,Y 508.053,Z 857.545,A -85,B 0,C 180,E1 23631.5,E2 23631.5} C_VEL
LIN {X 0,Y 508.968,Z 838.584,A -85,B 0,C 180,E1 23630.914,E2 23630.914} C_VEL
LIN {X 0,Y 509.83,Z 813.721,A -85,B 0,C 180,E1 23630.355,E2 23630.355} C_VEL
LIN {X 0,Y 512.527,Z 609.591,A -85,B 0,C 180,E1 23627.156,E2 23627.156} C_VEL
LIN {X 0,Y 514.401,Z 486.054,A -85,B 0,C 180,E1 23625.107,E2 23625.107} C_VEL
LIN {X 0,Y 511.788,Z 465.187,A -85,B 0,C 180,E1 23624.457,E2 23624.457} C_VEL
LIN {X 0,Y 513.276,Z 432.642,A -85,B 0,C 180,E1 23622.603,E2 23622.603} C_VEL
LIN {X 0,Y 502.586,Z 411.916,A -85,B 0,C 180,E1 23620.133,E2 23620.133} C_VEL
LIN {X 0,Y 495.991,Z 399.76,A -85,B 0,C 180,E1 23618.528,E2 23618.528} C_VEL
LIN {X 0,Y 491.536,Z 391.504,A -85,B 0,C 180,E1 23617.386,E2 23617.386} C_VEL
LIN {X 0,Y 489.114,Z 387.744,A -85,B 0,C 180,E1 23616.795,E2 23616.795} C_VEL
LIN {X 0,Y 488.76,Z 386.227,A -85,B 0,C 180,E1 23616.502,E2 23616.502} C_VEL
LIN {X 0,Y 488.769,Z 386.166,A -85,B 0,C 180,E1 23612.966,E2 23612.966} C_VEL
LIN {X 0,Y 488.805,Z 386.138,A -85,B 0,C 180,E1 23609.535,E2 23609.535} C_VEL
LIN {X 0,Y 488.75,Z 386.134,A -85,B 0,C 180,E1 23606.092,E2 23606.092} C_VEL
LIN {X 0,Y 488.779,Z 386.164,A -85,B 0,C 180,E1 23602.617,E2 23602.617} C_VEL
LIN {X 0,Y 488.775,Z 386.124,A -85,B 0,C 180,E1 23599.353,E2 23599.353} C_VEL
LIN {X 0,Y 488.755,Z 386.163,A -85,B 0,C 180,E1 23595.91,E2 23595.91} C_VEL
LIN {X 0,Y 488.811,Z 386.118,A -85,B 0,C 180,E1 23592.522,E2 23592.522} C_VEL
LIN {X 0,Y 488.768,Z 386.162,A -85,B 0,C 180,E1 23589.062,E2 23589.062} C_VEL
LIN {X 0,Y 488.758,Z 386.16,A -85,B 0,C 180,E1 23585.517,E2 23585.517} C_VEL
LIN {X 0,Y 488.819,Z 386.159,A -85,B 0,C 180,E1 23582.11,E2 23582.11} C_VEL
LIN {X 0,Y 488.764,Z 386.162,A -85,B 0,C 180,E1 23578.71,E2 23578.71} C_VEL
LIN {X 0,Y 488.761,Z 386.162,A -85,B 0,C 180,E1 23575.071,E2 23575.071} C_VEL
LIN {X 0,Y 488.824,Z 386.154,A -85,B 0,C 180,E1 23571.649,E2 23571.649} C_VEL
LIN {X 0,Y 488.769,Z 386.154,A -85,B 0,C 180,E1 23568.196,E2 23568.196} C_VEL
LIN {X 0,Y 488.766,Z 386.157,A -85,B 0,C 180,E1 23564.698,E2 23564.698} C_VEL
LIN {X 0,Y 488.822,Z 386.15,A -85,B 0,C 180,E1 23561.268,E2 23561.268} C_VEL
LIN {X 0,Y 488.763,Z 386.155,A -85,B 0,C 180,E1 23557.888,E2 23557.888} C_VEL
LIN {X 0,Y 488.77,Z 386.156,A -85,B 0,C 180,E1 23554.298,E2 23554.298} C_VEL
LIN {X 0,Y 488.83,Z 386.126,A -85,B 0,C 180,E1 23550.856,E2 23550.856} C_VEL
LIN {X 0,Y 488.768,Z 386.16,A -85,B 0,C 180,E1 23547.44,E2 23547.44} C_VEL
LIN {X 0,Y 488.772,Z 386.127,A -85,B 0,C 180,E1 23543.903,E2 23543.903} C_VEL
LIN {X 0,Y 488.826,Z 386.144,A -85,B 0,C 180,E1 23540.456,E2 23540.456} C_VEL
LIN {X 0,Y 488.767,Z 386.162,A -85,B 0,C 180,E1 23537.061,E2 23537.061} C_VEL
LIN {X 0,Y 488.856,Z 386.391,A -85,B 0,C 180,E1 23534.173,E2 23534.173} C_VEL
LIN {X 0,Y 490.312,Z 389.937,A -85,B 0,C 180,E1 23533.572,E2 23533.572} C_VEL
LIN {X 0,Y 495.212,Z 399.589,A -85,B 0,C 180,E1 23532.011,E2 23532.011} C_VEL
LIN {X 0,Y 502.823,Z 415.884,A -85,B 0,C 180,E1 23529.597,E2 23529.597} C_VEL
LIN {X 0,Y 506.892,Z 425.293,A -85,B 0,C 180,E1 23528.307,E2 23528.307} C_VEL
LIN {X 0,Y 506.114,Z 435.006,A -85,B 0,C 180,E1 23527.531,E2 23527.531} C_VEL
LIN {X 0,Y 504.818,Z 441.599,A -85,B 0,C 180,E1 23527.09,E2 23527.09} C_VEL
LIN {X 0,Y 498.48,Z 460.124,A -85,B 0,C 180,E1 23526.142,E2 23526.142} C_VEL
LIN {X 0,Y 497.475,Z 465.791,A -85,B 0,C 180,E1 23525.756,E2 23525.756} C_VEL
LIN {X 0,Y 497.362,Z 470.422,A -85,B 0,C 180,E1 23525.431,E2 23525.431} C_VEL
LIN {X 0,Y 501.015,Z 492.07,A -85,B 0,C 180,E1 23524.699,E2 23524.699} C_VEL
LIN {X 0,Y 497.921,Z 727.682,A -85,B 0,C 180,E1 23521.124,E2 23521.124} C_VEL
LIN {X 0,Y 497.379,Z 747.806,A -85,B 0,C 180,E1 23520.699,E2 23520.699} C_VEL
LIN {X 0,Y 496.426,Z 767.042,A -85,B 0,C 180,E1 23520.088,E2 23520.088} C_VEL
LIN {X 0,Y 495.071,Z 786.492,A -85,B 0,C 180,E1 23519.252,E2 23519.252} C_VEL
LIN {X 0,Y 493.589,Z 803.905,A -85,B 0,C 180,E1 23518.295,E2 23518.295} C_VEL
LIN {X 0,Y 491.752,Z 821.47,A -85,B 0,C 180,E1 23517.094,E2 23517.094} C_VEL
LIN {X 0,Y 489.815,Z 838.194,A -85,B 0,C 180,E1 23515.708,E2 23515.708} C_VEL
LIN {X 0,Y 487.8,Z 854.626,A -85,B 0,C 180,E1 23514.073,E2 23514.073} C_VEL
LIN {X 0,Y 485.849,Z 870,A -85,B 0,C 180,E1 23512.251,E2 23512.251} C_VEL
LIN {X 0,Y 484.176,Z 883.831,A -85,B 0,C 180,E1 23510.3,E2 23510.3} C_VEL
LIN {X 0,Y 482.746,Z 896.287,A -85,B 0,C 180,E1 23508.225,E2 23508.225} C_VEL
LIN {X 0,Y 481.559,Z 907.881,A -85,B 0,C 180,E1 23505.907,E2 23505.907} C_VEL
LIN {X 0,Y 480.749,Z 917.432,A -85,B 0,C 180,E1 23503.593,E2 23503.593} C_VEL
LIN {X 0,Y 480.256,Z 927.341,A -85,B 0,C 180,E1 23500.8,E2 23500.8} C_VEL
LIN {X 0,Y 480.04,Z 934,A -85,B 0,C 180,E1 23498.384,E2 23498.384} C_VEL
LIN {X 0,Y 479.949,Z 938.889,A -85,B 0,C 180,E1 23495.979,E2 23495.979} C_VEL
LIN {X 0,Y 479.906,Z 942.234,A -85,B 0,C 180,E1 23493.464,E2 23493.464} C_VEL
LIN {X 0,Y 479.907,Z 943.793,A -85,B 0,C 180,E1 23491.074,E2 23491.074} C_VEL
LIN {X 0,Y 479.902,Z 943.766,A -85,B 0,C 180,E1 23488.687,E2 23488.687} C_VEL
LIN {X 0,Y 479.91,Z 942.094,A -85,B 0,C 180,E1 23486.297,E2 23486.297} C_VEL
LIN {X 0,Y 479.951,Z 938.836,A -85,B 0,C 180,E1 23483.901,E2 23483.901} C_VEL
LIN {X 0,Y 480.048,Z 933.922,A -85,B 0,C 180,E1 23481.496,E2 23481.496} C_VEL
LIN {X 0,Y 480.258,Z 927.24,A -85,B 0,C 180,E1 23479.079,E2 23479.079} C_VEL
LIN {X 0,Y 480.756,Z 917.307,A -85,B 0,C 180,E1 23476.285,E2 23476.285} C_VEL
LIN {X 0,Y 481.571,Z 907.721,A -85,B 0,C 180,E1 23473.97,E2 23473.97} C_VEL
LIN {X 0,Y 482.767,Z 896.094,A -85,B 0,C 180,E1 23471.651,E2 23471.651} C_VEL
LIN {X 0,Y 484.318,Z 882.834,A -85,B 0,C 180,E1 23469.454,E2 23469.454} C_VEL
LIN {X 0,Y 486.063,Z 868.495,A -85,B 0,C 180,E1 23467.462,E2 23467.462} C_VEL
LIN {X 0,Y 487.986,Z 853.193,A -85,B 0,C 180,E1 23465.679,E2 23465.679} C_VEL
LIN {X 0,Y 489.945,Z 837.124,A -85,B 0,C 180,E1 23464.105,E2 23464.105} C_VEL
LIN {X 0,Y 491.983,Z 819.318,A -85,B 0,C 180,E1 23462.658,E2 23462.658} C_VEL
LIN {X 0,Y 493.753,Z 802.066,A -85,B 0,C 180,E1 23461.505,E2 23461.505} C_VEL
LIN {X 0,Y 495.357,Z 783.218,A -85,B 0,C 180,E1 23460.494,E2 23460.494} C_VEL
LIN {X 0,Y 496.595,Z 764.439,A -85,B 0,C 180,E1 23459.726,E2 23459.726} C_VEL
LIN {X 0,Y 497.49,Z 744.238,A -85,B 0,C 180,E1 23459.121,E2 23459.121} C_VEL
LIN {X 0,Y 498.026,Z 720.638,A -85,B 0,C 180,E1 23458.675,E2 23458.675} C_VEL
LIN {X 0,Y 501.007,Z 491.37,A -85,B 0,C 180,E1 23455.198,E2 23455.198} C_VEL
LIN {X 0,Y 497.258,Z 468.933,A -85,B 0,C 180,E1 23454.401,E2 23454.401} C_VEL
LIN {X 0,Y 500.376,Z 428.98,A -85,B 0,C 180,E1 23451.225,E2 23451.225} C_VEL
LIN {X 0,Y 492.664,Z 411.632,A -85,B 0,C 180,E1 23448.731,E2 23448.731} C_VEL
LIN {X 0,Y 486.765,Z 399.579,A -85,B 0,C 180,E1 23446.82,E2 23446.82} C_VEL
LIN {X 0,Y 482.686,Z 391.292,A -85,B 0,C 180,E1 23445.445,E2 23445.445} C_VEL
LIN {X 0,Y 480.973,Z 387.919,A -85,B 0,C 180,E1 23444.856,E2 23444.856} C_VEL
LIN {X 0,Y 480.84,Z 387.146,A -85,B 0,C 180,E1 23444.563,E2 23444.563} C_VEL
LIN {X 0,Y 480.834,Z 387.116,A -85,B 0,C 180,E1 23440.921,E2 23440.921} C_VEL
LIN {X 0,Y 480.89,Z 387.13,A -85,B 0,C 180,E1 23437.532,E2 23437.532} C_VEL
LIN {X 0,Y 480.846,Z 387.145,A -85,B 0,C 180,E1 23433.935,E2 23433.935} C_VEL
LIN {X 0,Y 480.826,Z 387.11,A -85,B 0,C 180,E1 23430.347,E2 23430.347} C_VEL
LIN {X 0,Y 480.879,Z 387.149,A -85,B 0,C 180,E1 23426.875,E2 23426.875} C_VEL
LIN {X 0,Y 480.851,Z 387.15,A -85,B 0,C 180,E1 23423.401,E2 23423.401} C_VEL
LIN {X 0,Y 480.83,Z 387.151,A -85,B 0,C 180,E1 23419.94,E2 23419.94} C_VEL
LIN {X 0,Y 480.878,Z 387.148,A -85,B 0,C 180,E1 23416.426,E2 23416.426} C_VEL
LIN {X 0,Y 480.844,Z 387.15,A -85,B 0,C 180,E1 23412.978,E2 23412.978} C_VEL
LIN {X 0,Y 480.827,Z 387.152,A -85,B 0,C 180,E1 23409.456,E2 23409.456} C_VEL
LIN {X 0,Y 480.886,Z 387.144,A -85,B 0,C 180,E1 23406.087,E2 23406.087} C_VEL
LIN {X 0,Y 480.834,Z 387.145,A -85,B 0,C 180,E1 23402.622,E2 23402.622} C_VEL
LIN {X 0,Y 480.824,Z 387.149,A -85,B 0,C 180,E1 23399.047,E2 23399.047} C_VEL
LIN {X 0,Y 480.875,Z 387.139,A -85,B 0,C 180,E1 23395.588,E2 23395.588} C_VEL
LIN {X 0,Y 480.828,Z 387.141,A -85,B 0,C 180,E1 23392.232,E2 23392.232} C_VEL
LIN {X 0,Y 480.819,Z 387.135,A -85,B 0,C 180,E1 23388.607,E2 23388.607} C_VEL
LIN {X 0,Y 480.881,Z 387.125,A -85,B 0,C 180,E1 23385.183,E2 23385.183} C_VEL
LIN {X 0,Y 480.829,Z 387.125,A -85,B 0,C 180,E1 23381.7,E2 23381.7} C_VEL
LIN {X 0,Y 480.819,Z 387.15,A -85,B 0,C 180,E1 23378.147,E2 23378.147} C_VEL
LIN {X 0,Y 480.871,Z 387.11,A -85,B 0,C 180,E1 23374.754,E2 23374.754} C_VEL
LIN {X 0,Y 480.826,Z 387.151,A -85,B 0,C 180,E1 23371.292,E2 23371.292} C_VEL
LIN {X 0,Y 480.815,Z 387.139,A -85,B 0,C 180,E1 23367.695,E2 23367.695} C_VEL
LIN {X 0,Y 480.895,Z 387.311,A -85,B 0,C 180,E1 23364.471,E2 23364.471} C_VEL
LIN {X 0,Y 481.096,Z 388.256,A -85,B 0,C 180,E1 23364.268,E2 23364.268} C_VEL
LIN {X 0,Y 482.65,Z 391.293,A -85,B 0,C 180,E1 23363.815,E2 23363.815} C_VEL
LIN {X 0,Y 483.861,Z 393.273,A -85,B 0,C 180,E1 23363.499,E2 23363.499} C_VEL
LIN {X 0,Y 489.018,Z 402.264,A -85,B 0,C 180,E1 23362.166,E2 23362.166} C_VEL
LIN {X 0,Y 498.347,Z 419.382,A -85,B 0,C 180,E1 23359.856,E2 23359.856} C_VEL
LIN {X 0,Y 507.045,Z 436.717,A -85,B 0,C 180,E1 23357.784,E2 23357.784} C_VEL
LIN {X 0,Y 505.54,Z 466.619,A -85,B 0,C 180,E1 23356.086,E2 23356.086} C_VEL
LIN {X 0,Y 508.29,Z 489.857,A -85,B 0,C 180,E1 23355.386,E2 23355.386} C_VEL
LIN {X 0,Y 505.156,Z 666.229,A -85,B 0,C 180,E1 23352.457,E2 23352.457} C_VEL
LIN {X 0,Y 502.888,Z 816.578,A -85,B 0,C 180,E1 23350.057,E2 23350.057} C_VEL
LIN {X 0,Y 501.931,Z 839.581,A -85,B 0,C 180,E1 23349.505,E2 23349.505} C_VEL
LIN {X 0,Y 500.79,Z 862.07,A -85,B 0,C 180,E1 23348.787,E2 23348.787} C_VEL
LIN {X 0,Y 499.248,Z 885.142,A -85,B 0,C 180,E1 23347.831,E2 23347.831} C_VEL
LIN {X 0,Y 497.814,Z 904.659,A -85,B 0,C 180,E1 23346.837,E2 23346.837} C_VEL
LIN {X 0,Y 495.821,Z 924.118,A -85,B 0,C 180,E1 23345.576,E2 23345.576} C_VEL
LIN {X 0,Y 493.623,Z 944.166,A -85,B 0,C 180,E1 23344.061,E2 23344.061} C_VEL
LIN {X 0,Y 491.392,Z 963.256,A -85,B 0,C 180,E1 23342.354,E2 23342.354} C_VEL
LIN {X 0,Y 489.089,Z 982.78,A -85,B 0,C 180,E1 23340.328,E2 23340.328} C_VEL
LIN {X 0,Y 487.199,Z 999.148,A -85,B 0,C 180,E1 23338.366,E2 23338.366} C_VEL
LIN {X 0,Y 485.37,Z 1015.136,A -85,B 0,C 180,E1 23336.158,E2 23336.158} C_VEL
LIN {X 0,Y 483.888,Z 1029.505,A -85,B 0,C 180,E1 23333.891,E2 23333.891} C_VEL
LIN {X 0,Y 482.622,Z 1042.447,A -85,B 0,C 180,E1 23331.512,E2 23331.512} C_VEL
LIN {X 0,Y 481.596,Z 1054.769,A -85,B 0,C 180,E1 23328.898,E2 23328.898} C_VEL
LIN {X 0,Y 480.903,Z 1064.606,A -85,B 0,C 180,E1 23326.425,E2 23326.425} C_VEL
LIN {X 0,Y 480.406,Z 1073.637,A -85,B 0,C 180,E1 23323.725,E2 23323.725} C_VEL
LIN {X 0,Y 480.133,Z 1080.388,A -85,B 0,C 180,E1 23321.237,E2 23321.237} C_VEL
LIN {X 0,Y 479.99,Z 1086.428,A -85,B 0,C 180,E1 23318.385,E2 23318.385} C_VEL
LIN {X 0,Y 479.913,Z 1090.278,A -85,B 0,C 180,E1 23315.859,E2 23315.859} C_VEL
LIN {X 0,Y 479.886,Z 1092.918,A -85,B 0,C 180,E1 23313.105,E2 23313.105} C_VEL
LIN {X 0,Y 479.884,Z 1093.872,A -85,B 0,C 180,E1 23310.716,E2 23310.716} C_VEL
LIN {X 0,Y 479.907,Z 1093.594,A -85,B 0,C 180,E1 23308.09,E2 23308.09} C_VEL
LIN {X 0,Y 479.908,Z 1091.728,A -85,B 0,C 180,E1 23305.459,E2 23305.459} C_VEL
LIN {X 0,Y 479.925,Z 1088.494,A -85,B 0,C 180,E1 23302.819,E2 23302.819} C_VEL
LIN {X 0,Y 480.021,Z 1083.827,A -85,B 0,C 180,E1 23300.287,E2 23300.287} C_VEL
LIN {X 0,Y 480.239,Z 1077.826,A -85,B 0,C 180,E1 23297.739,E2 23297.739} C_VEL
LIN {X 0,Y 480.62,Z 1069.745,A -85,B 0,C 180,E1 23295.051,E2 23295.051} C_VEL
LIN {X 0,Y 481.204,Z 1060.444,A -85,B 0,C 180,E1 23292.465,E2 23292.465} C_VEL
LIN {X 0,Y 482.056,Z 1049.149,A -85,B 0,C 180,E1 23289.86,E2 23289.86} C_VEL
LIN {X 0,Y 483.253,Z 1035.85,A -85,B 0,C 180,E1 23287.238,E2 23287.238} C_VEL
LIN {X 0,Y 484.63,Z 1022.211,A -85,B 0,C 180,E1 23284.919,E2 23284.919} C_VEL
LIN {X 0,Y 486.298,Z 1006.763,A -85,B 0,C 180,E1 23282.649,E2 23282.649} C_VEL
LIN {X 0,Y 488.285,Z 989.927,A -85,B 0,C 180,E1 23280.489,E2 23280.489} C_VEL
LIN {X 0,Y 490.333,Z 972.166,A -85,B 0,C 180,E1 23278.532,E2 23278.532} C_VEL
LIN {X 0,Y 492.684,Z 952.243,A -85,B 0,C 180,E1 23276.635,E2 23276.635} C_VEL
LIN {X 0,Y 494.772,Z 933.693,A -85,B 0,C 180,E1 23275.117,E2 23275.117} C_VEL
LIN {X 0,Y 496.993,Z 912.813,A -85,B 0,C 180,E1 23273.666,E2 23273.666} C_VEL
LIN {X 0,Y 498.405,Z 897.16,A -85,B 0,C 180,E1 23272.758,E2 23272.758} C_VEL
LIN {X 0,Y 499.902,Z 876.574,A -85,B 0,C 180,E1 23271.786,E2 23271.786} C_VEL
LIN {X 0,Y 501.226,Z 853.407,A -85,B 0,C 180,E1 23270.918,E2 23270.918} C_VEL
LIN {X 0,Y 502.366,Z 829.445,A -85,B 0,C 180,E1 23270.226,E2 23270.226} C_VEL
LIN {X 0,Y 503.137,Z 806.716,A -85,B 0,C 180,E1 23269.77,E2 23269.77} C_VEL
LIN {X 0,Y 505.826,Z 621.306,A -85,B 0,C 180,E1 23266.818,E2 23266.818} C_VEL
LIN {X 0,Y 508.19,Z 487.551,A -85,B 0,C 180,E1 23264.561,E2 23264.561} C_VEL
LIN {X 0,Y 505.484,Z 465.188,A -85,B 0,C 180,E1 23263.855,E2 23263.855} C_VEL
LIN {X 0,Y 506.931,Z 436.494,A -85,B 0,C 180,E1 23262.19,E2 23262.19} C_VEL
LIN {X 0,Y 496.812,Z 416.7,A -85,B 0,C 180,E1 23259.791,E2 23259.791} C_VEL
LIN {X 0,Y 490.257,Z 404.673,A -85,B 0,C 180,E1 23258.166,E2 23258.166} C_VEL
LIN {X 0,Y 485.571,Z 396.294,A -85,B 0,C 180,E1 23256.96,E2 23256.96} C_VEL
LIN {X 0,Y 483.108,Z 391.81,A -85,B 0,C 180,E1 23256.293,E2 23256.293} C_VEL
LIN {X 0,Y 481.224,Z 388.696,A -85,B 0,C 180,E1 23255.794,E2 23255.794} C_VEL
LIN {X 0,Y 480.879,Z 387.219,A -85,B 0,C 180,E1 23255.494,E2 23255.494} C_VEL
LIN {X 0,Y 480.827,Z 387.131,A -85,B 0,C 180,E1 23252.023,E2 23252.023} C_VEL
LIN {X 0,Y 480.816,Z 387.156,A -85,B 0,C 180,E1 23248.437,E2 23248.437} C_VEL
LIN {X 0,Y 480.861,Z 387.114,A -85,B 0,C 180,E1 23244.962,E2 23244.962} C_VEL
LIN {X 0,Y 480.828,Z 387.142,A -85,B 0,C 180,E1 23241.596,E2 23241.596} C_VEL
LIN {X 0,Y 480.816,Z 387.134,A -85,B 0,C 180,E1 23238.05,E2 23238.05} C_VEL
LIN {X 0,Y 480.871,Z 387.123,A -85,B 0,C 180,E1 23234.571,E2 23234.571} C_VEL
LIN {X 0,Y 480.828,Z 387.133,A -85,B 0,C 180,E1 23231.15,E2 23231.15} C_VEL
LIN {X 0,Y 480.82,Z 387.14,A -85,B 0,C 180,E1 23227.648,E2 23227.648} C_VEL
LIN {X 0,Y 480.876,Z 387.137,A -85,B 0,C 180,E1 23224.292,E2 23224.292} C_VEL
LIN {X 0,Y 480.823,Z 387.147,A -85,B 0,C 180,E1 23220.834,E2 23220.834} C_VEL
LIN {X 0,Y 480.825,Z 387.146,A -85,B 0,C 180,E1 23217.258,E2 23217.258} C_VEL
LIN {X 0,Y 480.886,Z 387.142,A -85,B 0,C 180,E1 23213.793,E2 23213.793} C_VEL
LIN {X 0,Y 480.825,Z 387.152,A -85,B 0,C 180,E1 23210.424,E2 23210.424} C_VEL
LIN {X 0,Y 480.826,Z 387.152,A -85,B 0,C 180,E1 23206.777,E2 23206.777} C_VEL
LIN {X 0,Y 480.883,Z 387.149,A -85,B 0,C 180,E1 23203.441,E2 23203.441} C_VEL
LIN {X 0,Y 480.83,Z 387.151,A -85,B 0,C 180,E1 23199.933,E2 23199.933} C_VEL
LIN {X 0,Y 480.83,Z 387.152,A -85,B 0,C 180,E1 23196.338,E2 23196.338} C_VEL
LIN {X 0,Y 480.89,Z 387.148,A -85,B 0,C 180,E1 23192.86,E2 23192.86} C_VEL
LIN {X 0,Y 480.827,Z 387.111,A -85,B 0,C 180,E1 23189.418,E2 23189.418} C_VEL
LIN {X 0,Y 480.829,Z 387.146,A -85,B 0,C 180,E1 23185.843,E2 23185.843} C_VEL
LIN {X 0,Y 480.88,Z 387.133,A -85,B 0,C 180,E1 23182.317,E2 23182.317} C_VEL
LIN {X 0,Y 480.834,Z 387.116,A -85,B 0,C 180,E1 23178.921,E2 23178.921} C_VEL
LIN {X 0,Y 480.833,Z 387.187,A -85,B 0,C 180,E1 23175.268,E2 23175.268} C_VEL
LIN {X 0,Y 481.125,Z 388.514,A -85,B 0,C 180,E1 23174.958,E2 23174.958} C_VEL
LIN {X 0,Y 483.249,Z 392.247,A -85,B 0,C 180,E1 23174.284,E2 23174.284} C_VEL
LIN {X 0,Y 491.544,Z 409.291,A -85,B 0,C 180,E1 23171.534,E2 23171.534} C_VEL
LIN {X 0,Y 499.586,Z 427.146,A -85,B 0,C 180,E1 23168.935,E2 23168.935} C_VEL
LIN {X 0,Y 500.364,Z 429.425,A -85,B 0,C 180,E1 23168.643,E2 23168.643} C_VEL
LIN {X 0,Y 497.475,Z 465.791,A -85,B 0,C 180,E1 23165.756,E2 23165.756} C_VEL
LIN {X 0,Y 497.993,Z 471.767,A -85,B 0,C 180,E1 23165.37,E2 23165.37} C_VEL
LIN {X 0,Y 499.011,Z 478.22,A -85,B 0,C 180,E1 23165.132,E2 23165.132} C_VEL
LIN {X 0,Y 498.841,Z 483.905,A -85,B 0,C 180,E1 23165.055,E2 23165.055} C_VEL
LIN {X 0,Y 495.161,Z 497.649,A -85,B 0,C 180,E1 23165.184,E2 23165.184} C_VEL
LIN {X 0,Y 494.79,Z 501.147,A -85,B 0,C 180,E1 23165.159,E2 23165.159} C_VEL
LIN {X 0,Y 491.691,Z 737.083,A -85,B 0,C 180,E1 23161.565,E2 23161.565} C_VEL
LIN {X 0,Y 490.966,Z 757.015,A -85,B 0,C 180,E1 23161.06,E2 23161.06} C_VEL
LIN {X 0,Y 489.814,Z 776.609,A -85,B 0,C 180,E1 23160.346,E2 23160.346} C_VEL
LIN {X 0,Y 488.421,Z 794.251,A -85,B 0,C 180,E1 23159.501,E2 23159.501} C_VEL
LIN {X 0,Y 486.619,Z 811.925,A -85,B 0,C 180,E1 23158.428,E2 23158.428} C_VEL
LIN {X 0,Y 484.591,Z 829.343,A -85,B 0,C 180,E1 23157.129,E2 23157.129} C_VEL
LIN {X 0,Y 482.446,Z 845.918,A -85,B 0,C 180,E1 23155.64,E2 23155.64} C_VEL
LIN {X 0,Y 480.329,Z 861.609,A -85,B 0,C 180,E1 23153.949,E2 23153.949} C_VEL
LIN {X 0,Y 478.204,Z 876.922,A -85,B 0,C 180,E1 23151.979,E2 23151.979} C_VEL
LIN {X 0,Y 476.251,Z 891.305,A -85,B 0,C 180,E1 23149.756,E2 23149.756} C_VEL
LIN {X 0,Y 474.7,Z 903.928,A -85,B 0,C 180,E1 23147.403,E2 23147.403} C_VEL
LIN {X 0,Y 473.494,Z 914.893,A -85,B 0,C 180,E1 23144.929,E2 23144.929} C_VEL
LIN {X 0,Y 472.717,Z 923.766,A -85,B 0,C 180,E1 23142.459,E2 23142.459} C_VEL
LIN {X 0,Y 472.227,Z 930.826,A -85,B 0,C 180,E1 23139.999,E2 23139.999} C_VEL
LIN {X 0,Y 471.982,Z 936.729,A -85,B 0,C 180,E1 23137.302,E2 23137.302} C_VEL
LIN {X 0,Y 471.926,Z 940.866,A -85,B 0,C 180,E1 23134.74,E2 23134.74} C_VEL
LIN {X 0,Y 471.912,Z 943.276,A -85,B 0,C 180,E1 23132.186,E2 23132.186} C_VEL
LIN {X 0,Y 471.906,Z 943.97,A -85,B 0,C 180,E1 23129.757,E2 23129.757} C_VEL
LIN {X 0,Y 471.907,Z 943.056,A -85,B 0,C 180,E1 23127.328,E2 23127.328} C_VEL
LIN {X 0,Y 471.923,Z 940.506,A -85,B 0,C 180,E1 23124.895,E2 23124.895} C_VEL
LIN {X 0,Y 472.014,Z 935.954,A -85,B 0,C 180,E1 23122.208,E2 23122.208} C_VEL
LIN {X 0,Y 472.261,Z 930.093,A -85,B 0,C 180,E1 23119.633,E2 23119.633} C_VEL
LIN {X 0,Y 472.829,Z 922.399,A -85,B 0,C 180,E1 23117.047,E2 23117.047} C_VEL
LIN {X 0,Y 473.645,Z 913.181,A -85,B 0,C 180,E1 23114.574,E2 23114.574} C_VEL
LIN {X 0,Y 474.79,Z 903.116,A -85,B 0,C 180,E1 23112.347,E2 23112.347} C_VEL
LIN {X 0,Y 476.283,Z 891.092,A -85,B 0,C 180,E1 23110.118,E2 23110.118} C_VEL
LIN {X 0,Y 478.241,Z 876.661,A -85,B 0,C 180,E1 23107.894,E2 23107.894} C_VEL
LIN {X 0,Y 480.299,Z 861.81,A -85,B 0,C 180,E1 23105.985,E2 23105.985} C_VEL
LIN {X 0,Y 482.366,Z 846.5,A -85,B 0,C 180,E1 23104.328,E2 23104.328} C_VEL
LIN {X 0,Y 484.471,Z 830.365,A -85,B 0,C 180,E1 23102.864,E2 23102.864} C_VEL
LIN {X 0,Y 486.468,Z 813.521,A -85,B 0,C 180,E1 23101.588,E2 23101.588} C_VEL
LIN {X 0,Y 488.262,Z 795.835,A -85,B 0,C 180,E1 23100.495,E2 23100.495} C_VEL
LIN {X 0,Y 489.737,Z 777.789,A -85,B 0,C 180,E1 23099.614,E2 23099.614} C_VEL
LIN {X 0,Y 490.926,Z 757.958,A -85,B 0,C 180,E1 23098.877,E2 23098.877} C_VEL
LIN {X 0,Y 491.68,Z 738.094,A -85,B 0,C 180,E1 23098.363,E2 23098.363} C_VEL
LIN {X 0,Y 493.185,Z 618.25,A -85,B 0,C 180,E1 23096.527,E2 23096.527} C_VEL
LIN {X 0,Y 494.781,Z 491.88,A -85,B 0,C 180,E1 23094.59,E2 23094.59} C_VEL
LIN {X 0,Y 490.909,Z 469.058,A -85,B 0,C 180,E1 23093.761,E2 23093.761} C_VEL
LIN {X 0,Y 493.867,Z 432.735,A -85,B 0,C 180,E1 23090.842,E2 23090.842} C_VEL
LIN {X 0,Y 486.508,Z 416.131,A -85,B 0,C 180,E1 23088.408,E2 23088.408} C_VEL
LIN {X 0,Y 479.368,Z 401.258,A -85,B 0,C 180,E1 23086.007,E2 23086.007} C_VEL
LIN {X 0,Y 476.757,Z 396.348,A -85,B 0,C 180,E1 23085.142,E2 23085.142} C_VEL
LIN {X 0,Y 474.577,Z 392.095,A -85,B 0,C 180,E1 23084.385,E2 23084.385} C_VEL
LIN {X 0,Y 472.988,Z 388.411,A -85,B 0,C 180,E1 23083.7,E2 23083.7} C_VEL
LIN {X 0,Y 472.894,Z 388.106,A -85,B 0,C 180,E1 23080.433,E2 23080.433} C_VEL
LIN {X 0,Y 472.895,Z 388.106,A -85,B 0,C 180,E1 23076.742,E2 23076.742} C_VEL
LIN {X 0,Y 472.946,Z 388.138,A -85,B 0,C 180,E1 23073.2,E2 23073.2} C_VEL
LIN {X 0,Y 472.911,Z 388.096,A -85,B 0,C 180,E1 23069.653,E2 23069.653} C_VEL
LIN {X 0,Y 472.893,Z 388.135,A -85,B 0,C 180,E1 23066.09,E2 23066.09} C_VEL
LIN {X 0,Y 472.933,Z 388.129,A -85,B 0,C 180,E1 23062.63,E2 23062.63} C_VEL
LIN {X 0,Y 472.916,Z 388.133,A -85,B 0,C 180,E1 23059.13,E2 23059.13} C_VEL
LIN {X 0,Y 472.887,Z 388.135,A -85,B 0,C 180,E1 23055.577,E2 23055.577} C_VEL
LIN {X 0,Y 472.92,Z 388.131,A -85,B 0,C 180,E1 23052.082,E2 23052.082} C_VEL
LIN {X 0,Y 472.918,Z 388.139,A -85,B 0,C 180,E1 23048.634,E2 23048.634} C_VEL
LIN {X 0,Y 472.884,Z 388.141,A -85,B 0,C 180,E1 23045.095,E2 23045.095} C_VEL
LIN {X 0,Y 472.913,Z 388.14,A -85,B 0,C 180,E1 23041.575,E2 23041.575} C_VEL
LIN {X 0,Y 472.915,Z 388.137,A -85,B 0,C 180,E1 23038.183,E2 23038.183} C_VEL
LIN {X 0,Y 472.882,Z 388.141,A -85,B 0,C 180,E1 23034.662,E2 23034.662} C_VEL
LIN {X 0,Y 472.92,Z 388.135,A -85,B 0,C 180,E1 23031.245,E2 23031.245} C_VEL
LIN {X 0,Y 472.902,Z 388.099,A -85,B 0,C 180,E1 23027.794,E2 23027.794} C_VEL
LIN {X 0,Y 472.88,Z 388.14,A -85,B 0,C 180,E1 23024.298,E2 23024.298} C_VEL
LIN {X 0,Y 472.92,Z 388.094,A -85,B 0,C 180,E1 23020.871,E2 23020.871} C_VEL
LIN {X 0,Y 472.902,Z 388.141,A -85,B 0,C 180,E1 23017.369,E2 23017.369} C_VEL
LIN {X 0,Y 472.874,Z 388.106,A -85,B 0,C 180,E1 23013.909,E2 23013.909} C_VEL
LIN {X 0,Y 472.931,Z 388.111,A -85,B 0,C 180,E1 23010.489,E2 23010.489} C_VEL
LIN {X 0,Y 472.888,Z 388.145,A -85,B 0,C 180,E1 23007.078,E2 23007.078} C_VEL
LIN {X 0,Y 472.899,Z 388.307,A -85,B 0,C 180,E1 23005.547,E2 23005.547} C_VEL
LIN {X 0,Y 473.374,Z 390.065,A -85,B 0,C 180,E1 23005.23,E2 23005.23} C_VEL
LIN {X 0,Y 475.897,Z 393.901,A -85,B 0,C 180,E1 23004.559,E2 23004.559} C_VEL
LIN {X 0,Y 477.893,Z 397.551,A -85,B 0,C 180,E1 23003.991,E2 23003.991} C_VEL
LIN {X 0,Y 484.164,Z 408.733,A -85,B 0,C 180,E1 23002.319,E2 23002.319} C_VEL
LIN {X 0,Y 491.593,Z 422.473,A -85,B 0,C 180,E1 23000.431,E2 23000.431} C_VEL
LIN {X 0,Y 500.713,Z 440.515,A -85,B 0,C 180,E1 22998.207,E2 22998.207} C_VEL
LIN {X 0,Y 499.291,Z 466.755,A -85,B 0,C 180,E1 22996.696,E2 22996.696} C_VEL
LIN {X 0,Y 502.092,Z 491.309,A -85,B 0,C 180,E1 22995.943,E2 22995.943} C_VEL
LIN {X 0,Y 498.316,Z 680.603,A -85,B 0,C 180,E1 22992.74,E2 22992.74} C_VEL
LIN {X 0,Y 496.022,Z 816.05,A -85,B 0,C 180,E1 22990.54,E2 22990.54} C_VEL
LIN {X 0,Y 494.991,Z 839.125,A -85,B 0,C 180,E1 22989.977,E2 22989.977} C_VEL
LIN {X 0,Y 493.716,Z 862.109,A -85,B 0,C 180,E1 22989.225,E2 22989.225} C_VEL
LIN {X 0,Y 492.134,Z 884.292,A -85,B 0,C 180,E1 22988.292,E2 22988.292} C_VEL
LIN {X 0,Y 490.302,Z 908.087,A -85,B 0,C 180,E1 22987.057,E2 22987.057} C_VEL
LIN {X 0,Y 488.566,Z 927.999,A -85,B 0,C 180,E1 22985.825,E2 22985.825} C_VEL
LIN {X 0,Y 486.612,Z 945.635,A -85,B 0,C 180,E1 22984.478,E2 22984.478} C_VEL
LIN {X 0,Y 484.354,Z 963.635,A -85,B 0,C 180,E1 22982.842,E2 22982.842} C_VEL
LIN {X 0,Y 481.9,Z 983.026,A -85,B 0,C 180,E1 22980.799,E2 22980.799} C_VEL
LIN {X 0,Y 479.818,Z 999.654,A -85,B 0,C 180,E1 22978.775,E2 22978.775} C_VEL
LIN {X 0,Y 477.901,Z 1015.135,A -85,B 0,C 180,E1 22976.598,E2 22976.598} C_VEL
LIN {X 0,Y 476.281,Z 1029.504,A -85,B 0,C 180,E1 22974.297,E2 22974.297} C_VEL
LIN {X 0,Y 474.849,Z 1042.914,A -85,B 0,C 180,E1 22971.786,E2 22971.786} C_VEL
LIN {X 0,Y 473.727,Z 1055.291,A -85,B 0,C 180,E1 22969.096,E2 22969.096} C_VEL
LIN {X 0,Y 472.982,Z 1065.064,A -85,B 0,C 180,E1 22966.582,E2 22966.582} C_VEL
LIN {X 0,Y 472.428,Z 1074.3,A -85,B 0,C 180,E1 22963.729,E2 22963.729} C_VEL
LIN {X 0,Y 472.145,Z 1080.865,A -85,B 0,C 180,E1 22961.235,E2 22961.235} C_VEL
LIN {X 0,Y 471.994,Z 1086.642,A -85,B 0,C 180,E1 22958.401,E2 22958.401} C_VEL
LIN {X 0,Y 471.914,Z 1090.438,A -85,B 0,C 180,E1 22955.837,E2 22955.837} C_VEL
LIN {X 0,Y 471.887,Z 1092.986,A -85,B 0,C 180,E1 22953.036,E2 22953.036} C_VEL
LIN {X 0,Y 471.885,Z 1093.872,A -85,B 0,C 180,E1 22950.728,E2 22950.728} C_VEL
LIN {X 0,Y 471.908,Z 1093.594,A -85,B 0,C 180,E1 22948.057,E2 22948.057} C_VEL
LIN {X 0,Y 471.908,Z 1091.728,A -85,B 0,C 180,E1 22945.382,E2 22945.382} C_VEL
LIN {X 0,Y 471.931,Z 1088.494,A -85,B 0,C 180,E1 22942.697,E2 22942.697} C_VEL
LIN {X 0,Y 472.035,Z 1083.827,A -85,B 0,C 180,E1 22940.121,E2 22940.121} C_VEL
LIN {X 0,Y 472.274,Z 1077.826,A -85,B 0,C 180,E1 22937.529,E2 22937.529} C_VEL
LIN {X 0,Y 472.7,Z 1069.744,A -85,B 0,C 180,E1 22934.794,E2 22934.794} C_VEL
LIN {X 0,Y 473.344,Z 1060.444,A -85,B 0,C 180,E1 22932.164,E2 22932.164} C_VEL
LIN {X 0,Y 474.274,Z 1049.147,A -85,B 0,C 180,E1 22929.515,E2 22929.515} C_VEL
LIN {X 0,Y 475.586,Z 1035.848,A -85,B 0,C 180,E1 22926.85,E2 22926.85} C_VEL
LIN {X 0,Y 477.05,Z 1022.57,A -85,B 0,C 180,E1 22924.554,E2 22924.554} C_VEL
LIN {X 0,Y 478.936,Z 1006.493,A -85,B 0,C 180,E1 22922.154,E2 22922.154} C_VEL
LIN {X 0,Y 481.052,Z 989.926,A -85,B 0,C 180,E1 22920,E2 22920} C_VEL
LIN {X 0,Y 483.275,Z 972.164,A -85,B 0,C 180,E1 22918.018,E2 22918.018} C_VEL
LIN {X 0,Y 485.795,Z 952.24,A -85,B 0,C 180,E1 22916.098,E2 22916.098} C_VEL
LIN {X 0,Y 487.725,Z 936.015,A -85,B 0,C 180,E1 22914.754,E2 22914.754} C_VEL
LIN {X 0,Y 489.258,Z 920.016,A -85,B 0,C 180,E1 22913.654,E2 22913.654} C_VEL
LIN {X 0,Y 491.163,Z 897.408,A -85,B 0,C 180,E1 22912.359,E2 22912.359} C_VEL
LIN {X 0,Y 492.841,Z 875.435,A -85,B 0,C 180,E1 22911.307,E2 22911.307} C_VEL
LIN {X 0,Y 494.276,Z 852.006,A -85,B 0,C 180,E1 22910.421,E2 22910.421} C_VEL
LIN {X 0,Y 495.528,Z 827.748,A -85,B 0,C 180,E1 22909.722,E2 22909.722} C_VEL
LIN {X 0,Y 496.321,Z 805.164,A -85,B 0,C 180,E1 22909.268,E2 22909.268} C_VEL
LIN {X 0,Y 499.223,Z 628.874,A -85,B 0,C 180,E1 22906.401,E2 22906.401} C_VEL
LIN {X 0,Y 502.006,Z 489.052,A -85,B 0,C 180,E1 22904.006,E2 22904.006} C_VEL
LIN {X 0,Y 499.239,Z 465.059,A -85,B 0,C 180,E1 22903.231,E2 22903.231} C_VEL
LIN {X 0,Y 500.596,Z 440.276,A -85,B 0,C 180,E1 22901.767,E2 22901.767} C_VEL
LIN {X 0,Y 490.428,Z 420.145,A -85,B 0,C 180,E1 22899.274,E2 22899.274} C_VEL
LIN {X 0,Y 480.805,Z 402.559,A -85,B 0,C 180,E1 22896.791,E2 22896.791} C_VEL
LIN {X 0,Y 475.879,Z 393.875,A -85,B 0,C 180,E1 22895.443,E2 22895.443} C_VEL
LIN {X 0,Y 473.224,Z 389.657,A -85,B 0,C 180,E1 22894.723,E2 22894.723} C_VEL
LIN {X 0,Y 472.881,Z 388.188,A -85,B 0,C 180,E1 22894.412,E2 22894.412} C_VEL
LIN {X 0,Y 472.88,Z 388.104,A -85,B 0,C 180,E1 22890.776,E2 22890.776} C_VEL
LIN {X 0,Y 472.935,Z 388.124,A -85,B 0,C 180,E1 22887.307,E2 22887.307} C_VEL
LIN {X 0,Y 472.882,Z 388.128,A -85,B 0,C 180,E1 22883.819,E2 22883.819} C_VEL
LIN {X 0,Y 472.875,Z 388.101,A -85,B 0,C 180,E1 22880.147,E2 22880.147} C_VEL
LIN {X 0,Y 472.937,Z 388.137,A -85,B 0,C 180,E1 22876.709,E2 22876.709} C_VEL
LIN {X 0,Y 472.88,Z 388.095,A -85,B 0,C 180,E1 22873.324,E2 22873.324} C_VEL
LIN {X 0,Y 472.882,Z 388.139,A -85,B 0,C 180,E1 22869.738,E2 22869.738} C_VEL
LIN {X 0,Y 472.945,Z 388.133,A -85,B 0,C 180,E1 22866.311,E2 22866.311} C_VEL
LIN {X 0,Y 472.892,Z 388.136,A -85,B 0,C 180,E1 22862.787,E2 22862.787} C_VEL
LIN {X 0,Y 472.883,Z 388.139,A -85,B 0,C 180,E1 22859.273,E2 22859.273} C_VEL
LIN {X 0,Y 472.933,Z 388.13,A -85,B 0,C 180,E1 22855.756,E2 22855.756} C_VEL
LIN {X 0,Y 472.892,Z 388.129,A -85,B 0,C 180,E1 22852.345,E2 22852.345} C_VEL
LIN {X 0,Y 472.884,Z 388.129,A -85,B 0,C 180,E1 22848.783,E2 22848.783} C_VEL
LIN {X 0,Y 472.939,Z 388.126,A -85,B 0,C 180,E1 22845.303,E2 22845.303} C_VEL
LIN {X 0,Y 472.903,Z 388.132,A -85,B 0,C 180,E1 22841.765,E2 22841.765} C_VEL
LIN {X 0,Y 472.885,Z 388.133,A -85,B 0,C 180,E1 22838.283,E2 22838.283} C_VEL
LIN {X 0,Y 472.934,Z 388.128,A -85,B 0,C 180,E1 22834.806,E2 22834.806} C_VEL
LIN {X 0,Y 472.906,Z 388.115,A -85,B 0,C 180,E1 22831.318,E2 22831.318} C_VEL
LIN {X 0,Y 472.886,Z 388.132,A -85,B 0,C 180,E1 22827.753,E2 22827.753} C_VEL
LIN {X 0,Y 472.925,Z 388.097,A -85,B 0,C 180,E1 22824.278,E2 22824.278} C_VEL
LIN {X 0,Y 472.913,Z 388.131,A -85,B 0,C 180,E1 22820.79,E2 22820.79} C_VEL
LIN {X 0,Y 472.887,Z 388.128,A -85,B 0,C 180,E1 22817.256,E2 22817.256} C_VEL
LIN {X 0,Y 472.98,Z 388.378,A -85,B 0,C 180,E1 22816.21,E2 22816.21} C_VEL
LIN {X 0,Y 474.329,Z 391.776,A -85,B 0,C 180,E1 22815.586,E2 22815.586} C_VEL
LIN {X 0,Y 475.466,Z 393.764,A -85,B 0,C 180,E1 22815.213,E2 22815.213} C_VEL
LIN {X 0,Y 478.097,Z 398.945,A -85,B 0,C 180,E1 22814.308,E2 22814.308} C_VEL
LIN {X 0,Y 484.039,Z 410.979,A -85,B 0,C 180,E1 22812.31,E2 22812.31} C_VEL
LIN {X 0,Y 491.151,Z 426.398,A -85,B 0,C 180,E1 22809.963,E2 22809.963} C_VEL
LIN {X 0,Y 493.894,Z 433.168,A -85,B 0,C 180,E1 22809.021,E2 22809.021} C_VEL
LIN {X 0,Y 490.95,Z 469.973,A -85,B 0,C 180,E1 22806.097,E2 22806.097} C_VEL
LIN {X 0,Y 494.911,Z 493.534,A -85,B 0,C 180,E1 22805.279,E2 22805.279} C_VEL
LIN {X 0,Y 494.79,Z 501.147,A -85,B 0,C 180,E1 22805.159,E2 22805.159} C_VEL
LIN {X 0,Y 493.935,Z 508.853,A -85,B 0,C 180,E1 22805.113,E2 22805.113} C_VEL
LIN {X 0,Y 488.857,Z 529.448,A -85,B 0,C 180,E1 22805.275,E2 22805.275} C_VEL
LIN {X 0,Y 488.183,Z 536.065,A -85,B 0,C 180,E1 22805.231,E2 22805.231} C_VEL
LIN {X 0,Y 485.495,Z 739.049,A -85,B 0,C 180,E1 22802.132,E2 22802.132} C_VEL
LIN {X 0,Y 484.756,Z 758.89,A -85,B 0,C 180,E1 22801.621,E2 22801.621} C_VEL
LIN {X 0,Y 483.602,Z 778.38,A -85,B 0,C 180,E1 22800.904,E2 22800.904} C_VEL
LIN {X 0,Y 482.188,Z 796.134,A -85,B 0,C 180,E1 22800.051,E2 22800.051} C_VEL
LIN {X 0,Y 480.304,Z 814.167,A -85,B 0,C 180,E1 22798.947,E2 22798.947} C_VEL
LIN {X 0,Y 478.187,Z 831.177,A -85,B 0,C 180,E1 22797.658,E2 22797.658} C_VEL
LIN {X 0,Y 475.824,Z 847.968,A -85,B 0,C 180,E1 22796.119,E2 22796.119} C_VEL
LIN {X 0,Y 473.5,Z 863.702,A -85,B 0,C 180,E1 22794.383,E2 22794.383} C_VEL
LIN {X 0,Y 471.255,Z 878.412,A -85,B 0,C 180,E1 22792.452,E2 22792.452} C_VEL
LIN {X 0,Y 469.097,Z 892.7,A -85,B 0,C 180,E1 22790.2,E2 22790.2} C_VEL
LIN {X 0,Y 467.357,Z 905.245,A -85,B 0,C 180,E1 22787.814,E2 22787.814} C_VEL
LIN {X 0,Y 465.98,Z 916.15,A -85,B 0,C 180,E1 22785.303,E2 22785.303} C_VEL
LIN {X 0,Y 465.077,Z 924.99,A -85,B 0,C 180,E1 22782.794,E2 22782.794} C_VEL
LIN {X 0,Y 464.479,Z 932.042,A -85,B 0,C 180,E1 22780.292,E2 22780.292} C_VEL
LIN {X 0,Y 464.169,Z 937.674,A -85,B 0,C 180,E1 22777.675,E2 22777.675} C_VEL
LIN {X 0,Y 464.009,Z 941.619,A -85,B 0,C 180,E1 22775.069,E2 22775.069} C_VEL
LIN {X 0,Y 463.954,Z 943.951,A -85,B 0,C 180,E1 22772.47,E2 22772.47} C_VEL
LIN {X 0,Y 463.946,Z 944.72,A -85,B 0,C 180,E1 22769.877,E2 22769.877} C_VEL
LIN {X 0,Y 463.953,Z 943.876,A -85,B 0,C 180,E1 22767.282,E2 22767.282} C_VEL
LIN {X 0,Y 464.011,Z 941.437,A -85,B 0,C 180,E1 22764.683,E2 22764.683} C_VEL
LIN {X 0,Y 464.19,Z 937.378,A -85,B 0,C 180,E1 22762.076,E2 22762.076} C_VEL
LIN {X 0,Y 464.504,Z 931.63,A -85,B 0,C 180,E1 22759.457,E2 22759.457} C_VEL
LIN {X 0,Y 465.127,Z 924.456,A -85,B 0,C 180,E1 22756.955,E2 22756.955} C_VEL
LIN {X 0,Y 465.995,Z 915.996,A -85,B 0,C 180,E1 22754.57,E2 22754.57} C_VEL
LIN {X 0,Y 467.381,Z 905.06,A -85,B 0,C 180,E1 22752.058,E2 22752.058} C_VEL
LIN {X 0,Y 469.122,Z 892.555,A -85,B 0,C 180,E1 22749.684,E2 22749.684} C_VEL
LIN {X 0,Y 471.159,Z 878.991,A -85,B 0,C 180,E1 22747.543,E2 22747.543} C_VEL
LIN {X 0,Y 473.298,Z 864.896,A -85,B 0,C 180,E1 22745.673,E2 22745.673} C_VEL
LIN {X 0,Y 475.616,Z 849.396,A -85,B 0,C 180,E1 22743.936,E2 22743.936} C_VEL
LIN {X 0,Y 477.968,Z 832.919,A -85,B 0,C 180,E1 22742.396,E2 22742.396} C_VEL
LIN {X 0,Y 480.09,Z 816.318,A -85,B 0,C 180,E1 22741.107,E2 22741.107} C_VEL
LIN {X 0,Y 481.918,Z 798.626,A -85,B 0,C 180,E1 22739.999,E2 22739.999} C_VEL
LIN {X 0,Y 483.493,Z 780.012,A -85,B 0,C 180,E1 22739.076,E2 22739.076} C_VEL
LIN {X 0,Y 484.669,Z 761.079,A -85,B 0,C 180,E1 22738.356,E2 22738.356} C_VEL
LIN {X 0,Y 485.476,Z 740.754,A -85,B 0,C 180,E1 22737.811,E2 22737.811} C_VEL
LIN {X 0,Y 486.139,Z 692.024,A -85,B 0,C 180,E1 22737.039,E2 22737.039} C_VEL
LIN {X 0,Y 488.8,Z 493.771,A -85,B 0,C 180,E1 22734.01,E2 22734.01} C_VEL
LIN {X 0,Y 484.621,Z 469.198,A -85,B 0,C 180,E1 22733.102,E2 22733.102} C_VEL
LIN {X 0,Y 487.458,Z 436.599,A -85,B 0,C 180,E1 22730.466,E2 22730.466} C_VEL
LIN {X 0,Y 479.469,Z 418.589,A -85,B 0,C 180,E1 22727.757,E2 22727.757} C_VEL
LIN {X 0,Y 471.684,Z 402.56,A -85,B 0,C 180,E1 22725.073,E2 22725.073} C_VEL
LIN {X 0,Y 467.432,Z 394.071,A -85,B 0,C 180,E1 22723.534,E2 22723.534} C_VEL
LIN {X 0,Y 465.463,Z 391.092,A -85,B 0,C 180,E1 22722.903,E2 22722.903} C_VEL
LIN {X 0,Y 464.983,Z 389.299,A -85,B 0,C 180,E1 22722.545,E2 22722.545} C_VEL
LIN {X 0,Y 464.983,Z 389.115,A -85,B 0,C 180,E1 22719.212,E2 22719.212} C_VEL
LIN {X 0,Y 464.994,Z 389.083,A -85,B 0,C 180,E1 22715.629,E2 22715.629} C_VEL
LIN {X 0,Y 464.954,Z 389.119,A -85,B 0,C 180,E1 22712.23,E2 22712.23} C_VEL
LIN {X 0,Y 464.97,Z 389.1,A -85,B 0,C 180,E1 22708.655,E2 22708.655} C_VEL
LIN {X 0,Y 465.001,Z 389.115,A -85,B 0,C 180,E1 22705.143,E2 22705.143} C_VEL
LIN {X 0,Y 464.951,Z 389.12,A -85,B 0,C 180,E1 22701.709,E2 22701.709} C_VEL
LIN {X 0,Y 464.96,Z 389.122,A -85,B 0,C 180,E1 22698.039,E2 22698.039} C_VEL
LIN {X 0,Y 465.01,Z 389.114,A -85,B 0,C 180,E1 22694.444,E2 22694.444} C_VEL
LIN {X 0,Y 464.963,Z 389.115,A -85,B 0,C 180,E1 22690.909,E2 22690.909} C_VEL
LIN {X 0,Y 464.947,Z 389.118,A -85,B 0,C 180,E1 22687.29,E2 22687.29} C_VEL
LIN {X 0,Y 464.987,Z 389.116,A -85,B 0,C 180,E1 22683.823,E2 22683.823} C_VEL
LIN {X 0,Y 464.979,Z 389.119,A -85,B 0,C 180,E1 22680.247,E2 22680.247} C_VEL
LIN {X 0,Y 464.944,Z 389.125,A -85,B 0,C 180,E1 22676.672,E2 22676.672} C_VEL
LIN {X 0,Y 464.96,Z 389.121,A -85,B 0,C 180,E1 22673.084,E2 22673.084} C_VEL
LIN {X 0,Y 464.994,Z 389.119,A -85,B 0,C 180,E1 22669.594,E2 22669.594} C_VEL
LIN {X 0,Y 464.941,Z 389.087,A -85,B 0,C 180,E1 22666.063,E2 22666.063} C_VEL
LIN {X 0,Y 464.943,Z 389.117,A -85,B 0,C 180,E1 22662.349,E2 22662.349} C_VEL
LIN {X 0,Y 464.988,Z 389.099,A -85,B 0,C 180,E1 22658.824,E2 22658.824} C_VEL
LIN {X 0,Y 464.947,Z 389.096,A -85,B 0,C 180,E1 22655.458,E2 22655.458} C_VEL
LIN {X 0,Y 464.943,Z 389.134,A -85,B 0,C 180,E1 22651.849,E2 22651.849} C_VEL
LIN {X 0,Y 464.984,Z 389.092,A -85,B 0,C 180,E1 22648.354,E2 22648.354} C_VEL
LIN {X 0,Y 465.007,Z 389.297,A -85,B 0,C 180,E1 22646.676,E2 22646.676} C_VEL
LIN {X 0,Y 465.48,Z 391.042,A -85,B 0,C 180,E1 22646.346,E2 22646.346} C_VEL
LIN {X 0,Y 467.542,Z 394.081,A -85,B 0,C 180,E1 22645.776,E2 22645.776} C_VEL
LIN {X 0,Y 469.853,Z 398.373,A -85,B 0,C 180,E1 22645.08,E2 22645.08} C_VEL
LIN {X 0,Y 471.079,Z 400.393,A -85,B 0,C 180,E1 22644.739,E2 22644.739} C_VEL
LIN {X 0,Y 478.525,Z 413.489,A -85,B 0,C 180,E1 22642.704,E2 22642.704} C_VEL
LIN {X 0,Y 487.957,Z 431.202,A -85,B 0,C 180,E1 22640.26,E2 22640.26} C_VEL
LIN {X 0,Y 494.408,Z 444.596,A -85,B 0,C 180,E1 22638.616,E2 22638.616} C_VEL
LIN {X 0,Y 493.087,Z 466.796,A -85,B 0,C 180,E1 22637.326,E2 22637.326} C_VEL
LIN {X 0,Y 495.957,Z 492.682,A -85,B 0,C 180,E1 22636.517,E2 22636.517} C_VEL
LIN {X 0,Y 491.736,Z 683.125,A -85,B 0,C 180,E1 22633.237,E2 22633.237} C_VEL
LIN {X 0,Y 489.169,Z 815.331,A -85,B 0,C 180,E1 22631.034,E2 22631.034} C_VEL
LIN {X 0,Y 488.023,Z 838.943,A -85,B 0,C 180,E1 22630.444,E2 22630.444} C_VEL
LIN {X 0,Y 486.547,Z 863.364,A -85,B 0,C 180,E1 22629.619,E2 22629.619} C_VEL
LIN {X 0,Y 484.894,Z 885.552,A -85,B 0,C 180,E1 22628.667,E2 22628.667} C_VEL
LIN {X 0,Y 483.052,Z 907.708,A -85,B 0,C 180,E1 22627.485,E2 22627.485} C_VEL
LIN {X 0,Y 481.045,Z 929.556,A -85,B 0,C 180,E1 22626.105,E2 22626.105} C_VEL
LIN {X 0,Y 478.846,Z 950.641,A -85,B 0,C 180,E1 22624.517,E2 22624.517} C_VEL
LIN {X 0,Y 477.288,Z 964.485,A -85,B 0,C 180,E1 22623.296,E2 22623.296} C_VEL
LIN {X 0,Y 474.725,Z 983.388,A -85,B 0,C 180,E1 22621.27,E2 22621.27} C_VEL
LIN {X 0,Y 472.462,Z 1000.16,A -85,B 0,C 180,E1 22619.196,E2 22619.196} C_VEL
LIN {X 0,Y 470.351,Z 1015.978,A -85,B 0,C 180,E1 22616.923,E2 22616.923} C_VEL
LIN {X 0,Y 468.519,Z 1030.939,A -85,B 0,C 180,E1 22614.457,E2 22614.457} C_VEL
LIN {X 0,Y 467.056,Z 1043.713,A -85,B 0,C 180,E1 22612.002,E2 22612.002} C_VEL
LIN {X 0,Y 465.816,Z 1056.322,A -85,B 0,C 180,E1 22609.172,E2 22609.172} C_VEL
LIN {X 0,Y 465.033,Z 1065.98,A -85,B 0,C 180,E1 22606.616,E2 22606.616} C_VEL
LIN {X 0,Y 464.462,Z 1074.7,A -85,B 0,C 180,E1 22603.825,E2 22603.825} C_VEL
LIN {X 0,Y 464.153,Z 1081.47,A -85,B 0,C 180,E1 22601.179,E2 22601.179} C_VEL
LIN {X 0,Y 463.998,Z 1086.842,A -85,B 0,C 180,E1 22598.426,E2 22598.426} C_VEL
LIN {X 0,Y 463.915,Z 1090.597,A -85,B 0,C 180,E1 22595.814,E2 22595.814} C_VEL
LIN {X 0,Y 463.886,Z 1092.985,A -85,B 0,C 180,E1 22593.089,E2 22593.089} C_VEL
LIN {X 0,Y 463.885,Z 1093.872,A -85,B 0,C 180,E1 22590.741,E2 22590.741} C_VEL
LIN {X 0,Y 463.909,Z 1093.594,A -85,B 0,C 180,E1 22588.024,E2 22588.024} C_VEL
LIN {X 0,Y 463.909,Z 1091.841,A -85,B 0,C 180,E1 22585.426,E2 22585.426} C_VEL
LIN {X 0,Y 463.933,Z 1088.681,A -85,B 0,C 180,E1 22582.695,E2 22582.695} C_VEL
LIN {X 0,Y 464.044,Z 1084.082,A -85,B 0,C 180,E1 22580.074,E2 22580.074} C_VEL
LIN {X 0,Y 464.283,Z 1078.437,A -85,B 0,C 180,E1 22577.563,E2 22577.563} C_VEL
LIN {X 0,Y 464.758,Z 1070.148,A -85,B 0,C 180,E1 22574.656,E2 22574.656} C_VEL
LIN {X 0,Y 465.452,Z 1060.923,A -85,B 0,C 180,E1 22571.981,E2 22571.981} C_VEL
LIN {X 0,Y 466.453,Z 1049.719,A -85,B 0,C 180,E1 22569.287,E2 22569.287} C_VEL
LIN {X 0,Y 467.793,Z 1037.247,A -85,B 0,C 180,E1 22566.708,E2 22566.708} C_VEL
LIN {X 0,Y 469.398,Z 1023.613,A -85,B 0,C 180,E1 22564.292,E2 22564.292} C_VEL
LIN {X 0,Y 471.494,Z 1007.178,A -85,B 0,C 180,E1 22561.777,E2 22561.777} C_VEL
LIN {X 0,Y 473.775,Z 990.528,A -85,B 0,C 180,E1 22559.569,E2 22559.569} C_VEL
LIN {X 0,Y 476.137,Z 973.036,A -85,B 0,C 180,E1 22557.583,E2 22557.583} C_VEL
LIN {X 0,Y 477.881,Z 959.674,A -85,B 0,C 180,E1 22556.255,E2 22556.255} C_VEL
LIN {X 0,Y 479.858,Z 941.302,A -85,B 0,C 180,E1 22554.748,E2 22554.748} C_VEL
LIN {X 0,Y 481.852,Z 920.555,A -85,B 0,C 180,E1 22553.301,E2 22553.301} C_VEL
LIN {X 0,Y 483.993,Z 896.917,A -85,B 0,C 180,E1 22551.914,E2 22551.914} C_VEL
LIN {X 0,Y 485.587,Z 877.012,A -85,B 0,C 180,E1 22550.944,E2 22550.944} C_VEL
LIN {X 0,Y 487.183,Z 853.031,A -85,B 0,C 180,E1 22550.004,E2 22550.004} C_VEL
LIN {X 0,Y 488.535,Z 829.402,A -85,B 0,C 180,E1 22549.289,E2 22549.289} C_VEL
LIN {X 0,Y 489.458,Z 805.905,A -85,B 0,C 180,E1 22548.796,E2 22548.796} C_VEL
LIN {X 0,Y 492.715,Z 632.369,A -85,B 0,C 180,E1 22545.907,E2 22545.907} C_VEL
LIN {X 0,Y 495.864,Z 490.397,A -85,B 0,C 180,E1 22543.429,E2 22543.429} C_VEL
LIN {X 0,Y 493.043,Z 465.031,A -85,B 0,C 180,E1 22542.596,E2 22542.596} C_VEL
LIN {X 0,Y 494.303,Z 444.073,A -85,B 0,C 180,E1 22541.34,E2 22541.34} C_VEL
LIN {X 0,Y 484.894,Z 425.354,A -85,B 0,C 180,E1 22538.969,E2 22538.969} C_VEL
LIN {X 0,Y 475.583,Z 408.212,A -85,B 0,C 180,E1 22536.51,E2 22536.51} C_VEL
LIN {X 0,Y 470.293,Z 398.878,A -85,B 0,C 180,E1 22535.031,E2 22535.031} C_VEL
LIN {X 0,Y 468.236,Z 395.617,A -85,B 0,C 180,E1 22534.462,E2 22534.462} C_VEL
LIN {X 0,Y 467.514,Z 394.06,A -85,B 0,C 180,E1 22534.226,E2 22534.226} C_VEL
LIN {X 0,Y 465.456,Z 390.988,A -85,B 0,C 180,E1 22533.656,E2 22533.656} C_VEL
LIN {X 0,Y 465.036,Z 389.437,A -85,B 0,C 180,E1 22533.395,E2 22533.395} C_VEL
LIN {X 0,Y 464.934,Z 389.119,A -85,B 0,C 180,E1 22532.522,E2 22532.522} C_VEL
LIN {X 0,Y 464.976,Z 389.11,A -85,B 0,C 180,E1 22529.076,E2 22529.076} C_VEL
LIN {X 0,Y 464.958,Z 389.087,A -85,B 0,C 180,E1 22525.609,E2 22525.609} C_VEL
LIN {X 0,Y 464.939,Z 389.132,A -85,B 0,C 180,E1 22522.046,E2 22522.046} C_VEL
LIN {X 0,Y 464.962,Z 389.092,A -85,B 0,C 180,E1 22518.497,E2 22518.497} C_VEL
LIN {X 0,Y 464.969,Z 389.11,A -85,B 0,C 180,E1 22515.081,E2 22515.081} C_VEL
LIN {X 0,Y 464.936,Z 389.099,A -85,B 0,C 180,E1 22511.536,E2 22511.536} C_VEL
LIN {X 0,Y 464.966,Z 389.114,A -85,B 0,C 180,E1 22508.034,E2 22508.034} C_VEL
LIN {X 0,Y 464.977,Z 389.117,A -85,B 0,C 180,E1 22504.563,E2 22504.563} C_VEL
LIN {X 0,Y 464.941,Z 389.125,A -85,B 0,C 180,E1 22500.985,E2 22500.985} C_VEL
LIN {X 0,Y 464.956,Z 389.123,A -85,B 0,C 180,E1 22497.411,E2 22497.411} C_VEL
LIN {X 0,Y 465.006,Z 389.12,A -85,B 0,C 180,E1 22493.828,E2 22493.828} C_VEL
LIN {X 0,Y 464.951,Z 389.131,A -85,B 0,C 180,E1 22490.343,E2 22490.343} C_VEL
LIN {X 0,Y 464.946,Z 389.13,A -85,B 0,C 180,E1 22486.697,E2 22486.697} C_VEL
LIN {X 0,Y 465.002,Z 389.127,A -85,B 0,C 180,E1 22483.254,E2 22483.254} C_VEL
LIN {X 0,Y 464.972,Z 389.13,A -85,B 0,C 180,E1 22479.613,E2 22479.613} C_VEL
LIN {X 0,Y 464.946,Z 389.131,A -85,B 0,C 180,E1 22476.059,E2 22476.059} C_VEL
LIN {X 0,Y 464.973,Z 389.126,A -85,B 0,C 180,E1 22472.462,E2 22472.462} C_VEL
LIN {X 0,Y 464.976,Z 389.083,A -85,B 0,C 180,E1 22469.074,E2 22469.074} C_VEL
LIN {X 0,Y 464.947,Z 389.11,A -85,B 0,C 180,E1 22465.557,E2 22465.557} C_VEL
LIN {X 0,Y 464.964,Z 389.123,A -85,B 0,C 180,E1 22461.89,E2 22461.89} C_VEL
LIN {X 0,Y 464.996,Z 389.086,A -85,B 0,C 180,E1 22458.443,E2 22458.443} C_VEL
LIN {X 0,Y 464.984,Z 389.359,A -85,B 0,C 180,E1 22457.325,E2 22457.325} C_VEL
LIN {X 0,Y 466.351,Z 392.724,A -85,B 0,C 180,E1 22456.679,E2 22456.679} C_VEL
LIN {X 0,Y 467.574,Z 394.607,A -85,B 0,C 180,E1 22456.285,E2 22456.285} C_VEL
LIN {X 0,Y 474.044,Z 407.318,A -85,B 0,C 180,E1 22454.008,E2 22454.008} C_VEL
LIN {X 0,Y 481.716,Z 423.497,A -85,B 0,C 180,E1 22451.38,E2 22451.38} C_VEL
LIN {X 0,Y 487.448,Z 436.926,A -85,B 0,C 180,E1 22449.409,E2 22449.409} C_VEL
LIN {X 0,Y 484.672,Z 470.006,A -85,B 0,C 180,E1 22446.763,E2 22446.763} C_VEL
LIN {X 0,Y 488.858,Z 494.973,A -85,B 0,C 180,E1 22445.872,E2 22445.872} C_VEL
LIN {X 0,Y 488.183,Z 536.065,A -85,B 0,C 180,E1 22445.231,E2 22445.231} C_VEL
LIN {X 0,Y 487.307,Z 543.774,A -85,B 0,C 180,E1 22445.189,E2 22445.189} C_VEL
LIN {X 0,Y 482.225,Z 564.361,A -85,B 0,C 180,E1 22445.36,E2 22445.36} C_VEL
LIN {X 0,Y 481.562,Z 570.977,A -85,B 0,C 180,E1 22445.316,E2 22445.316} C_VEL
LIN {X 0,Y 479.271,Z 740.213,A -85,B 0,C 180,E1 22442.715,E2 22442.715} C_VEL
LIN {X 0,Y 478.502,Z 760.069,A -85,B 0,C 180,E1 22442.198,E2 22442.198} C_VEL
LIN {X 0,Y 477.317,Z 779.417,A -85,B 0,C 180,E1 22441.482,E2 22441.482} C_VEL
LIN {X 0,Y 475.874,Z 797.076,A -85,B 0,C 180,E1 22440.632,E2 22440.632} C_VEL
LIN {X 0,Y 473.918,Z 815.354,A -85,B 0,C 180,E1 22439.514,E2 22439.514} C_VEL
LIN {X 0,Y 471.738,Z 832.648,A -85,B 0,C 180,E1 22438.207,E2 22438.207} C_VEL
LIN {X 0,Y 469.38,Z 849.018,A -85,B 0,C 180,E1 22436.71,E2 22436.71} C_VEL
LIN {X 0,Y 467.079,Z 863.859,A -85,B 0,C 180,E1 22435.078,E2 22435.078} C_VEL
LIN {X 0,Y 464.626,Z 878.192,A -85,B 0,C 180,E1 22433.192,E2 22433.192} C_VEL
LIN {X 0,Y 462.334,Z 891.903,A -85,B 0,C 180,E1 22431.039,E2 22431.039} C_VEL
LIN {X 0,Y 460.379,Z 904.129,A -85,B 0,C 180,E1 22428.75,E2 22428.75} C_VEL
LIN {X 0,Y 458.744,Z 915.406,A -85,B 0,C 180,E1 22426.2,E2 22426.2} C_VEL
LIN {X 0,Y 457.624,Z 924.61,A -85,B 0,C 180,E1 22423.649,E2 22423.649} C_VEL
LIN {X 0,Y 456.831,Z 932.336,A -85,B 0,C 180,E1 22420.977,E2 22420.977} C_VEL
LIN {X 0,Y 456.407,Z 938.234,A -85,B 0,C 180,E1 22418.313,E2 22418.313} C_VEL
LIN {X 0,Y 456.183,Z 942.459,A -85,B 0,C 180,E1 22415.66,E2 22415.66} C_VEL
LIN {X 0,Y 456.085,Z 945.036,A -85,B 0,C 180,E1 22413.016,E2 22413.016} C_VEL
LIN {X 0,Y 456.056,Z 946.028,A -85,B 0,C 180,E1 22410.377,E2 22410.377} C_VEL
LIN {X 0,Y 456.072,Z 945.49,A -85,B 0,C 180,E1 22407.738,E2 22407.738} C_VEL
LIN {X 0,Y 456.146,Z 943.272,A -85,B 0,C 180,E1 22404.97,E2 22404.97} C_VEL
LIN {X 0,Y 456.331,Z 939.532,A -85,B 0,C 180,E1 22402.319,E2 22402.319} C_VEL
LIN {X 0,Y 456.691,Z 934.136,A -85,B 0,C 180,E1 22399.658,E2 22399.658} C_VEL
LIN {X 0,Y 457.388,Z 926.946,A -85,B 0,C 180,E1 22396.988,E2 22396.988} C_VEL
LIN {X 0,Y 458.455,Z 917.801,A -85,B 0,C 180,E1 22394.31,E2 22394.31} C_VEL
LIN {X 0,Y 459.988,Z 907.028,A -85,B 0,C 180,E1 22391.759,E2 22391.759} C_VEL
LIN {X 0,Y 461.786,Z 895.32,A -85,B 0,C 180,E1 22389.466,E2 22389.466} C_VEL
LIN {X 0,Y 463.958,Z 882.181,A -85,B 0,C 180,E1 22387.309,E2 22387.309} C_VEL
LIN {X 0,Y 466.266,Z 868.402,A -85,B 0,C 180,E1 22385.399,E2 22385.399} C_VEL
LIN {X 0,Y 468.722,Z 853.495,A -85,B 0,C 180,E1 22383.66,E2 22383.66} C_VEL
LIN {X 0,Y 471.13,Z 837.368,A -85,B 0,C 180,E1 22382.098,E2 22382.098} C_VEL
LIN {X 0,Y 473.26,Z 820.912,A -85,B 0,C 180,E1 22380.788,E2 22380.788} C_VEL
LIN {X 0,Y 475.267,Z 802.809,A -85,B 0,C 180,E1 22379.605,E2 22379.605} C_VEL
LIN {X 0,Y 476.973,Z 784.309,A -85,B 0,C 180,E1 22378.641,E2 22378.641} C_VEL
LIN {X 0,Y 478.268,Z 765.303,A -85,B 0,C 180,E1 22377.88,E2 22377.88} C_VEL
LIN {X 0,Y 479.098,Z 745.462,A -85,B 0,C 180,E1 22377.312,E2 22377.312} C_VEL
LIN {X 0,Y 479.588,Z 719.41,A -85,B 0,C 180,E1 22376.847,E2 22376.847} C_VEL
LIN {X 0,Y 482.851,Z 495.525,A -85,B 0,C 180,E1 22373.411,E2 22373.411} C_VEL
LIN {X 0,Y 478.406,Z 468.819,A -85,B 0,C 180,E1 22372.39,E2 22372.39} C_VEL
LIN {X 0,Y 481.068,Z 440.484,A -85,B 0,C 180,E1 22370.08,E2 22370.08} C_VEL
LIN {X 0,Y 473.536,Z 423.471,A -85,B 0,C 180,E1 22367.469,E2 22367.469} C_VEL
LIN {X 0,Y 466.228,Z 408.195,A -85,B 0,C 180,E1 22364.876,E2 22364.876} C_VEL
LIN {X 0,Y 461.589,Z 399.237,A -85,B 0,C 180,E1 22363.196,E2 22363.196} C_VEL
LIN {X 0,Y 459.673,Z 395.63,A -85,B 0,C 180,E1 22362.491,E2 22362.491} C_VEL
LIN {X 0,Y 457.263,Z 391.087,A -85,B 0,C 180,E1 22361.578,E2 22361.578} C_VEL
LIN {X 0,Y 457.045,Z 390.113,A -85,B 0,C 180,E1 22361.26,E2 22361.26} C_VEL
LIN {X 0,Y 457.07,Z 390.092,A -85,B 0,C 180,E1 22357.637,E2 22357.637} C_VEL
LIN {X 0,Y 457.025,Z 390.105,A -85,B 0,C 180,E1 22353.987,E2 22353.987} C_VEL
LIN {X 0,Y 457.009,Z 390.07,A -85,B 0,C 180,E1 22350.358,E2 22350.358} C_VEL
LIN {X 0,Y 457.053,Z 390.115,A -85,B 0,C 180,E1 22346.786,E2 22346.786} C_VEL
LIN {X 0,Y 457.052,Z 390.114,A -85,B 0,C 180,E1 22343.19,E2 22343.19} C_VEL
LIN {X 0,Y 457.013,Z 390.117,A -85,B 0,C 180,E1 22339.69,E2 22339.69} C_VEL
LIN {X 0,Y 457.023,Z 390.113,A -85,B 0,C 180,E1 22336.002,E2 22336.002} C_VEL
LIN {X 0,Y 457.066,Z 390.112,A -85,B 0,C 180,E1 22332.508,E2 22332.508} C_VEL
LIN {X 0,Y 457.019,Z 390.118,A -85,B 0,C 180,E1 22328.936,E2 22328.936} C_VEL
LIN {X 0,Y 457.009,Z 390.119,A -85,B 0,C 180,E1 22325.273,E2 22325.273} C_VEL
LIN {X 0,Y 457.051,Z 390.118,A -85,B 0,C 180,E1 22321.755,E2 22321.755} C_VEL
LIN {X 0,Y 457.032,Z 390.115,A -85,B 0,C 180,E1 22318.245,E2 22318.245} C_VEL
LIN {X 0,Y 457.006,Z 390.119,A -85,B 0,C 180,E1 22314.602,E2 22314.602} C_VEL
LIN {X 0,Y 457.017,Z 390.12,A -85,B 0,C 180,E1 22310.937,E2 22310.937} C_VEL
LIN {X 0,Y 457.058,Z 390.061,A -85,B 0,C 180,E1 22307.337,E2 22307.337} C_VEL
LIN {X 0,Y 457.013,Z 390.117,A -85,B 0,C 180,E1 22303.833,E2 22303.833} C_VEL
LIN {X 0,Y 456.998,Z 390.071,A -85,B 0,C 180,E1 22300.177,E2 22300.177} C_VEL
LIN {X 0,Y 457.046,Z 390.108,A -85,B 0,C 180,E1 22296.674,E2 22296.674} C_VEL
LIN {X 0,Y 457.031,Z 390.088,A -85,B 0,C 180,E1 22293.073,E2 22293.073} C_VEL
LIN {X 0,Y 456.994,Z 390.079,A -85,B 0,C 180,E1 22289.546,E2 22289.546} C_VEL
LIN {X 0,Y 457.036,Z 390.307,A -85,B 0,C 180,E1 22287.886,E2 22287.886} C_VEL
LIN {X 0,Y 457.318,Z 391.557,A -85,B 0,C 180,E1 22287.612,E2 22287.612} C_VEL
LIN {X 0,Y 459.219,Z 394.711,A -85,B 0,C 180,E1 22287.022,E2 22287.022} C_VEL
LIN {X 0,Y 460.088,Z 395.775,A -85,B 0,C 180,E1 22286.792,E2 22286.792} C_VEL
LIN {X 0,Y 461.922,Z 399.344,A -85,B 0,C 180,E1 22286.201,E2 22286.201} C_VEL
LIN {X 0,Y 463.137,Z 401.254,A -85,B 0,C 180,E1 22285.854,E2 22285.854} C_VEL
LIN {X 0,Y 468.345,Z 410.217,A -85,B 0,C 180,E1 22284.351,E2 22284.351} C_VEL
LIN {X 0,Y 477.498,Z 426.86,A -85,B 0,C 180,E1 22281.851,E2 22281.851} C_VEL
LIN {X 0,Y 486.906,Z 445.58,A -85,B 0,C 180,E1 22279.387,E2 22279.387} C_VEL
LIN {X 0,Y 488.102,Z 448.593,A -85,B 0,C 180,E1 22279.042,E2 22279.042} C_VEL
LIN {X 0,Y 486.943,Z 466.86,A -85,B 0,C 180,E1 22277.971,E2 22277.971} C_VEL
LIN {X 0,Y 489.878,Z 494.119,A -85,B 0,C 180,E1 22277.106,E2 22277.106} C_VEL
LIN {X 0,Y 484.916,Z 694.937,A -85,B 0,C 180,E1 22273.575,E2 22273.575} C_VEL
LIN {X 0,Y 482.361,Z 814.392,A -85,B 0,C 180,E1 22271.543,E2 22271.543} C_VEL
LIN {X 0,Y 481.13,Z 837.836,A -85,B 0,C 180,E1 22270.95,E2 22270.95} C_VEL
LIN {X 0,Y 479.55,Z 862.349,A -85,B 0,C 180,E1 22270.111,E2 22270.111} C_VEL
LIN {X 0,Y 477.835,Z 884.071,A -85,B 0,C 180,E1 22269.166,E2 22269.166} C_VEL
LIN {X 0,Y 475.817,Z 907.181,A -85,B 0,C 180,E1 22267.927,E2 22267.927} C_VEL
LIN {X 0,Y 473.79,Z 928.3,A -85,B 0,C 180,E1 22266.581,E2 22266.581} C_VEL
LIN {X 0,Y 471.511,Z 949.022,A -85,B 0,C 180,E1 22265.002,E2 22265.002} C_VEL
LIN {X 0,Y 469.254,Z 969.415,A -85,B 0,C 180,E1 22263.203,E2 22263.203} C_VEL
LIN {X 0,Y 467.534,Z 983.714,A -85,B 0,C 180,E1 22261.742,E2 22261.742} C_VEL
LIN {X 0,Y 465.747,Z 996.3,A -85,B 0,C 180,E1 22260.2,E2 22260.2} C_VEL
LIN {X 0,Y 463.42,Z 1012.595,A -85,B 0,C 180,E1 22257.917,E2 22257.917} C_VEL
LIN {X 0,Y 461.42,Z 1027.19,A -85,B 0,C 180,E1 22255.545,E2 22255.545} C_VEL
LIN {X 0,Y 459.675,Z 1041.171,A -85,B 0,C 180,E1 22252.914,E2 22252.914} C_VEL
LIN {X 0,Y 458.35,Z 1053.215,A -85,B 0,C 180,E1 22250.281,E2 22250.281} C_VEL
LIN {X 0,Y 457.346,Z 1063.685,A -85,B 0,C 180,E1 22247.56,E2 22247.56} C_VEL
LIN {X 0,Y 456.684,Z 1072.568,A -85,B 0,C 180,E1 22244.842,E2 22244.842} C_VEL
LIN {X 0,Y 456.267,Z 1079.652,A -85,B 0,C 180,E1 22242.144,E2 22242.144} C_VEL
LIN {X 0,Y 456.039,Z 1085.598,A -85,B 0,C 180,E1 22239.337,E2 22239.337} C_VEL
LIN {X 0,Y 455.943,Z 1089.799,A -85,B 0,C 180,E1 22236.548,E2 22236.548} C_VEL
LIN {X 0,Y 455.904,Z 1092.655,A -85,B 0,C 180,E1 22233.743,E2 22233.743} C_VEL
LIN {X 0,Y 455.893,Z 1093.826,A -85,B 0,C 180,E1 22231.005,E2 22231.005} C_VEL
LIN {X 0,Y 455.908,Z 1093.735,A -85,B 0,C 180,E1 22228.492,E2 22228.492} C_VEL
LIN {X 0,Y 455.911,Z 1092.068,A -85,B 0,C 180,E1 22225.598,E2 22225.598} C_VEL
LIN {X 0,Y 455.931,Z 1089.32,A -85,B 0,C 180,E1 22223.072,E2 22223.072} C_VEL
LIN {X 0,Y 456.047,Z 1084.59,A -85,B 0,C 180,E1 22220.153,E2 22220.153} C_VEL
LIN {X 0,Y 456.292,Z 1079.045,A -85,B 0,C 180,E1 22217.599,E2 22217.599} C_VEL
LIN {X 0,Y 456.79,Z 1070.957,A -85,B 0,C 180,E1 22214.642,E2 22214.642} C_VEL
LIN {X 0,Y 457.472,Z 1062.312,A -85,B 0,C 180,E1 22212.051,E2 22212.051} C_VEL
LIN {X 0,Y 458.579,Z 1050.864,A -85,B 0,C 180,E1 22209.182,E2 22209.182} C_VEL
LIN {X 0,Y 460.025,Z 1038.42,A -85,B 0,C 180,E1 22206.52,E2 22206.52} C_VEL
LIN {X 0,Y 461.803,Z 1024.315,A -85,B 0,C 180,E1 22203.964,E2 22203.964} C_VEL
LIN {X 0,Y 464.039,Z 1008.103,A -85,B 0,C 180,E1 22201.423,E2 22201.423} C_VEL
LIN {X 0,Y 466.324,Z 992.395,A -85,B 0,C 180,E1 22199.293,E2 22199.293} C_VEL
LIN {X 0,Y 468.246,Z 978.004,A -85,B 0,C 180,E1 22197.637,E2 22197.637} C_VEL
LIN {X 0,Y 470.411,Z 959.217,A -85,B 0,C 180,E1 22195.866,E2 22195.866} C_VEL
LIN {X 0,Y 472.846,Z 936.875,A -85,B 0,C 180,E1 22194.047,E2 22194.047} C_VEL
LIN {X 0,Y 474.95,Z 916.377,A -85,B 0,C 180,E1 22192.627,E2 22192.627} C_VEL
LIN {X 0,Y 477.01,Z 894.074,A -85,B 0,C 180,E1 22191.344,E2 22191.344} C_VEL
LIN {X 0,Y 478.813,Z 872.122,A -85,B 0,C 180,E1 22190.283,E2 22190.283} C_VEL
LIN {X 0,Y 480.464,Z 848.669,A -85,B 0,C 180,E1 22189.391,E2 22189.391} C_VEL
LIN {X 0,Y 481.9,Z 824.162,A -85,B 0,C 180,E1 22188.684,E2 22188.684} C_VEL
LIN {X 0,Y 482.811,Z 800.103,A -85,B 0,C 180,E1 22188.192,E2 22188.192} C_VEL
LIN {X 0,Y 485.925,Z 648.992,A -85,B 0,C 180,E1 22185.631,E2 22185.631} C_VEL
LIN {X 0,Y 489.799,Z 491.911,A -85,B 0,C 180,E1 22182.843,E2 22182.843} C_VEL
LIN {X 0,Y 486.88,Z 465.594,A -85,B 0,C 180,E1 22181.977,E2 22181.977} C_VEL
LIN {X 0,Y 487.981,Z 447.807,A -85,B 0,C 180,E1 22180.892,E2 22180.892} C_VEL
LIN {X 0,Y 479.141,Z 430.197,A -85,B 0,C 180,E1 22178.604,E2 22178.604} C_VEL
LIN {X 0,Y 470.36,Z 413.837,A -85,B 0,C 180,E1 22176.224,E2 22176.224} C_VEL
LIN {X 0,Y 464.663,Z 404.008,A -85,B 0,C 180,E1 22174.615,E2 22174.615} C_VEL
LIN {X 0,Y 462.328,Z 399.841,A -85,B 0,C 180,E1 22173.915,E2 22173.915} C_VEL
LIN {X 0,Y 460.364,Z 396.572,A -85,B 0,C 180,E1 22173.331,E2 22173.331} C_VEL
LIN {X 0,Y 459.646,Z 395.111,A -85,B 0,C 180,E1 22173.092,E2 22173.092} C_VEL
LIN {X 0,Y 457.501,Z 392.073,A -85,B 0,C 180,E1 22172.478,E2 22172.478} C_VEL
LIN {X 0,Y 457.037,Z 390.343,A -85,B 0,C 180,E1 22172.151,E2 22172.151} C_VEL
LIN {X 0,Y 457.05,Z 390.092,A -85,B 0,C 180,E1 22169.198,E2 22169.198} C_VEL
LIN {X 0,Y 457.015,Z 390.074,A -85,B 0,C 180,E1 22165.66,E2 22165.66} C_VEL
LIN {X 0,Y 457,Z 390.121,A -85,B 0,C 180,E1 22162.105,E2 22162.105} C_VEL
LIN {X 0,Y 457.035,Z 390.074,A -85,B 0,C 180,E1 22158.627,E2 22158.627} C_VEL
LIN {X 0,Y 457.029,Z 390.098,A -85,B 0,C 180,E1 22155.09,E2 22155.09} C_VEL
LIN {X 0,Y 456.997,Z 390.086,A -85,B 0,C 180,E1 22151.484,E2 22151.484} C_VEL
LIN {X 0,Y 457.009,Z 390.103,A -85,B 0,C 180,E1 22147.796,E2 22147.796} C_VEL
LIN {X 0,Y 457.056,Z 390.101,A -85,B 0,C 180,E1 22144.265,E2 22144.265} C_VEL
LIN {X 0,Y 457.012,Z 390.109,A -85,B 0,C 180,E1 22140.752,E2 22140.752} C_VEL
LIN {X 0,Y 457.004,Z 390.112,A -85,B 0,C 180,E1 22137.115,E2 22137.115} C_VEL
LIN {X 0,Y 457.049,Z 390.107,A -85,B 0,C 180,E1 22133.594,E2 22133.594} C_VEL
LIN {X 0,Y 457.032,Z 390.115,A -85,B 0,C 180,E1 22130.047,E2 22130.047} C_VEL
LIN {X 0,Y 457.004,Z 390.12,A -85,B 0,C 180,E1 22126.461,E2 22126.461} C_VEL
LIN {X 0,Y 457.035,Z 390.116,A -85,B 0,C 180,E1 22122.947,E2 22122.947} C_VEL
LIN {X 0,Y 457.068,Z 390.112,A -85,B 0,C 180,E1 22119.244,E2 22119.244} C_VEL
LIN {X 0,Y 457.014,Z 390.121,A -85,B 0,C 180,E1 22115.713,E2 22115.713} C_VEL
LIN {X 0,Y 457.011,Z 390.115,A -85,B 0,C 180,E1 22112.082,E2 22112.082} C_VEL
LIN {X 0,Y 457.058,Z 390.076,A -85,B 0,C 180,E1 22108.558,E2 22108.558} C_VEL
LIN {X 0,Y 457.026,Z 390.082,A -85,B 0,C 180,E1 22105.027,E2 22105.027} C_VEL
LIN {X 0,Y 457.01,Z 390.123,A -85,B 0,C 180,E1 22101.425,E2 22101.425} C_VEL
LIN {X 0,Y 457.057,Z 390.181,A -85,B 0,C 180,E1 22098.575,E2 22098.575} C_VEL
LIN {X 0,Y 457.482,Z 391.817,A -85,B 0,C 180,E1 22098.194,E2 22098.194} C_VEL
LIN {X 0,Y 459.631,Z 395.521,A -85,B 0,C 180,E1 22097.426,E2 22097.426} C_VEL
LIN {X 0,Y 461.56,Z 399.21,A -85,B 0,C 180,E1 22096.708,E2 22096.708} C_VEL
LIN {X 0,Y 468.532,Z 412.992,A -85,B 0,C 180,E1 22094.19,E2 22094.19} C_VEL
LIN {X 0,Y 475.947,Z 428.761,A -85,B 0,C 180,E1 22091.593,E2 22091.593} C_VEL
LIN {X 0,Y 481.028,Z 440.708,A -85,B 0,C 180,E1 22089.808,E2 22089.808} C_VEL
LIN {X 0,Y 478.443,Z 469.967,A -85,B 0,C 180,E1 22087.451,E2 22087.451} C_VEL
LIN {X 0,Y 482.855,Z 496.528,A -85,B 0,C 180,E1 22086.479,E2 22086.479} C_VEL
LIN {X 0,Y 481.562,Z 570.977,A -85,B 0,C 180,E1 22085.316,E2 22085.316} C_VEL
LIN {X 0,Y 480.697,Z 578.687,A -85,B 0,C 180,E1 22085.276,E2 22085.276} C_VEL
LIN {X 0,Y 475.629,Z 599.274,A -85,B 0,C 180,E1 22085.454,E2 22085.454} C_VEL
LIN {X 0,Y 474.972,Z 605.891,A -85,B 0,C 180,E1 22085.411,E2 22085.411} C_VEL
LIN {X 0,Y 473.055,Z 741.143,A -85,B 0,C 180,E1 22083.311,E2 22083.311} C_VEL
LIN {X 0,Y 472.245,Z 761.176,A -85,B 0,C 180,E1 22082.784,E2 22082.784} C_VEL
LIN {X 0,Y 470.993,Z 780.682,A -85,B 0,C 180,E1 22082.054,E2 22082.054} C_VEL
LIN {X 0,Y 469.431,Z 798.78,A -85,B 0,C 180,E1 22081.17,E2 22081.17} C_VEL
LIN {X 0,Y 467.398,Z 817.075,A -85,B 0,C 180,E1 22080.038,E2 22080.038} C_VEL
LIN {X 0,Y 465.222,Z 833.601,A -85,B 0,C 180,E1 22078.779,E2 22078.779} C_VEL
LIN {X 0,Y 462.658,Z 850.775,A -85,B 0,C 180,E1 22077.199,E2 22077.199} C_VEL
LIN {X 0,Y 460.169,Z 866.238,A -85,B 0,C 180,E1 22075.482,E2 22075.482} C_VEL
LIN {X 0,Y 457.779,Z 879.73,A -85,B 0,C 180,E1 22073.696,E2 22073.696} C_VEL
LIN {X 0,Y 455.451,Z 892.677,A -85,B 0,C 180,E1 22071.643,E2 22071.643} C_VEL
LIN {X 0,Y 453.264,Z 904.94,A -85,B 0,C 180,E1 22069.323,E2 22069.323} C_VEL
LIN {X 0,Y 451.416,Z 916.252,A -85,B 0,C 180,E1 22066.735,E2 22066.735} C_VEL
LIN {X 0,Y 450.108,Z 925.506,A -85,B 0,C 180,E1 22064.144,E2 22064.144} C_VEL
LIN {X 0,Y 449.214,Z 932.975,A -85,B 0,C 180,E1 22061.556,E2 22061.556} C_VEL
LIN {X 0,Y 448.675,Z 939.039,A -85,B 0,C 180,E1 22058.845,E2 22058.845} C_VEL
LIN {X 0,Y 448.366,Z 943.556,A -85,B 0,C 180,E1 22056.016,E2 22056.016} C_VEL
LIN {X 0,Y 448.214,Z 946.219,A -85,B 0,C 180,E1 22053.325,E2 22053.325} C_VEL
LIN {X 0,Y 448.175,Z 947.352,A -85,B 0,C 180,E1 22050.639,E2 22050.639} C_VEL
LIN {X 0,Y 448.195,Z 946.923,A -85,B 0,C 180,E1 22047.827,E2 22047.827} C_VEL
LIN {X 0,Y 448.281,Z 944.966,A -85,B 0,C 180,E1 22045.138,E2 22045.138} C_VEL
LIN {X 0,Y 448.494,Z 941.458,A -85,B 0,C 180,E1 22042.442,E2 22042.442} C_VEL
LIN {X 0,Y 448.918,Z 936.008,A -85,B 0,C 180,E1 22039.606,E2 22039.606} C_VEL
LIN {X 0,Y 449.737,Z 928.619,A -85,B 0,C 180,E1 22036.762,E2 22036.762} C_VEL
LIN {X 0,Y 450.926,Z 919.609,A -85,B 0,C 180,E1 22034.041,E2 22034.041} C_VEL
LIN {X 0,Y 452.609,Z 908.996,A -85,B 0,C 180,E1 22031.451,E2 22031.451} C_VEL
LIN {X 0,Y 454.578,Z 897.492,A -85,B 0,C 180,E1 22029.125,E2 22029.125} C_VEL
LIN {X 0,Y 456.921,Z 884.563,A -85,B 0,C 180,E1 22026.94,E2 22026.94} C_VEL
LIN {X 0,Y 459.408,Z 870.461,A -85,B 0,C 180,E1 22024.956,E2 22024.956} C_VEL
LIN {X 0,Y 461.889,Z 855.898,A -85,B 0,C 180,E1 22023.239,E2 22023.239} C_VEL
LIN {X 0,Y 464.369,Z 839.732,A -85,B 0,C 180,E1 22021.655,E2 22021.655} C_VEL
LIN {X 0,Y 466.598,Z 823.43,A -85,B 0,C 180,E1 22020.33,E2 22020.33} C_VEL
LIN {X 0,Y 468.705,Z 805.593,A -85,B 0,C 180,E1 22019.133,E2 22019.133} C_VEL
LIN {X 0,Y 470.543,Z 786.848,A -85,B 0,C 180,E1 22018.127,E2 22018.127} C_VEL
LIN {X 0,Y 471.91,Z 767.767,A -85,B 0,C 180,E1 22017.347,E2 22017.347} C_VEL
LIN {X 0,Y 472.833,Z 747.608,A -85,B 0,C 180,E1 22016.746,E2 22016.746} C_VEL
LIN {X 0,Y 473.355,Z 723.068,A -85,B 0,C 180,E1 22016.289,E2 22016.289} C_VEL
LIN {X 0,Y 476.927,Z 497.108,A -85,B 0,C 180,E1 22012.792,E2 22012.792} C_VEL
LIN {X 0,Y 472.247,Z 468.948,A -85,B 0,C 180,E1 22011.697,E2 22011.697} C_VEL
LIN {X 0,Y 474.609,Z 444.184,A -85,B 0,C 180,E1 22009.65,E2 22009.65} C_VEL
LIN {X 0,Y 467.578,Z 428.256,A -85,B 0,C 180,E1 22007.156,E2 22007.156} C_VEL
LIN {X 0,Y 460.509,Z 413.42,A -85,B 0,C 180,E1 22004.589,E2 22004.589} C_VEL
LIN {X 0,Y 455.783,Z 404.355,A -85,B 0,C 180,E1 22002.848,E2 22002.848} C_VEL
LIN {X 0,Y 453.359,Z 399.772,A -85,B 0,C 180,E1 22001.933,E2 22001.933} C_VEL
LIN {X 0,Y 451.404,Z 395.776,A -85,B 0,C 180,E1 22001.137,E2 22001.137} C_VEL
LIN {X 0,Y 449.548,Z 392.947,A -85,B 0,C 180,E1 22000.477,E2 22000.477} C_VEL
LIN {X 0,Y 449.127,Z 391.311,A -85,B 0,C 180,E1 22000.127,E2 22000.127} C_VEL
LIN {X 0,Y 449.073,Z 391.063,A -85,B 0,C 180,E1 21996.476,E2 21996.476} C_VEL
LIN {X 0,Y 449.092,Z 391.105,A -85,B 0,C 180,E1 21992.753,E2 21992.753} C_VEL
LIN {X 0,Y 449.134,Z 391.057,A -85,B 0,C 180,E1 21989.179,E2 21989.179} C_VEL
LIN {X 0,Y 449.088,Z 391.095,A -85,B 0,C 180,E1 21985.59,E2 21985.59} C_VEL
LIN {X 0,Y 449.074,Z 391.096,A -85,B 0,C 180,E1 21981.966,E2 21981.966} C_VEL
LIN {X 0,Y 449.111,Z 391.093,A -85,B 0,C 180,E1 21978.43,E2 21978.43} C_VEL
LIN {X 0,Y 449.106,Z 391.092,A -85,B 0,C 180,E1 21974.835,E2 21974.835} C_VEL
LIN {X 0,Y 449.07,Z 391.094,A -85,B 0,C 180,E1 21971.3,E2 21971.3} C_VEL
LIN {X 0,Y 449.075,Z 391.094,A -85,B 0,C 180,E1 21967.549,E2 21967.549} C_VEL
LIN {X 0,Y 449.118,Z 391.092,A -85,B 0,C 180,E1 21963.958,E2 21963.958} C_VEL
LIN {X 0,Y 449.099,Z 391.096,A -85,B 0,C 180,E1 21960.256,E2 21960.256} C_VEL
LIN {X 0,Y 449.067,Z 391.102,A -85,B 0,C 180,E1 21956.682,E2 21956.682} C_VEL
LIN {X 0,Y 449.076,Z 391.098,A -85,B 0,C 180,E1 21952.967,E2 21952.967} C_VEL
LIN {X 0,Y 449.117,Z 391.089,A -85,B 0,C 180,E1 21949.352,E2 21949.352} C_VEL
LIN {X 0,Y 449.085,Z 391.063,A -85,B 0,C 180,E1 21945.692,E2 21945.692} C_VEL
LIN {X 0,Y 449.061,Z 391.081,A -85,B 0,C 180,E1 21942.106,E2 21942.106} C_VEL
LIN {X 0,Y 449.077,Z 391.087,A -85,B 0,C 180,E1 21938.447,E2 21938.447} C_VEL
LIN {X 0,Y 449.106,Z 391.058,A -85,B 0,C 180,E1 21934.975,E2 21934.975} C_VEL
LIN {X 0,Y 449.068,Z 391.102,A -85,B 0,C 180,E1 21931.4,E2 21931.4} C_VEL
LIN {X 0,Y 449.086,Z 391.213,A -85,B 0,C 180,E1 21929.198,E2 21929.198} C_VEL
LIN {X 0,Y 449.329,Z 392.259,A -85,B 0,C 180,E1 21928.919,E2 21928.919} C_VEL
LIN {X 0,Y 451.094,Z 395.432,A -85,B 0,C 180,E1 21928.311,E2 21928.311} C_VEL
LIN {X 0,Y 452.261,Z 397.132,A -85,B 0,C 180,E1 21927.955,E2 21927.955} C_VEL
LIN {X 0,Y 454.515,Z 400.97,A -85,B 0,C 180,E1 21927.238,E2 21927.238} C_VEL
LIN {X 0,Y 461.525,Z 413.101,A -85,B 0,C 180,E1 21925.115,E2 21925.115} C_VEL
LIN {X 0,Y 468.435,Z 425.516,A -85,B 0,C 180,E1 21923.146,E2 21923.146} C_VEL
LIN {X 0,Y 477.259,Z 442.387,A -85,B 0,C 180,E1 21920.752,E2 21920.752} C_VEL
LIN {X 0,Y 481.835,Z 452.32,A -85,B 0,C 180,E1 21919.496,E2 21919.496} C_VEL
LIN {X 0,Y 480.864,Z 466.954,A -85,B 0,C 180,E1 21918.632,E2 21918.632} C_VEL
LIN {X 0,Y 483.852,Z 495.577,A -85,B 0,C 180,E1 21917.709,E2 21917.709} C_VEL
LIN {X 0,Y 478.315,Z 698.95,A -85,B 0,C 180,E1 21914.063,E2 21914.063} C_VEL
LIN {X 0,Y 475.565,Z 813.421,A -85,B 0,C 180,E1 21912.062,E2 21912.062} C_VEL
LIN {X 0,Y 474.183,Z 837.784,A -85,B 0,C 180,E1 21911.432,E2 21911.432} C_VEL
LIN {X 0,Y 472.463,Z 862.602,A -85,B 0,C 180,E1 21910.559,E2 21910.559} C_VEL
LIN {X 0,Y 470.593,Z 885.194,A -85,B 0,C 180,E1 21909.558,E2 21909.558} C_VEL
LIN {X 0,Y 468.457,Z 907.867,A -85,B 0,C 180,E1 21908.298,E2 21908.298} C_VEL
LIN {X 0,Y 466.074,Z 931.001,A -85,B 0,C 180,E1 21906.765,E2 21906.765} C_VEL
LIN {X 0,Y 463.821,Z 950.913,A -85,B 0,C 180,E1 21905.214,E2 21905.214} C_VEL
LIN {X 0,Y 461.469,Z 970.763,A -85,B 0,C 180,E1 21903.39,E2 21903.39} C_VEL
LIN {X 0,Y 459.131,Z 989.79,A -85,B 0,C 180,E1 21901.388,E2 21901.388} C_VEL
LIN {X 0,Y 457.284,Z 1004.234,A -85,B 0,C 180,E1 21899.614,E2 21899.614} C_VEL
LIN {X 0,Y 455.548,Z 1015.974,A -85,B 0,C 180,E1 21897.873,E2 21897.873} C_VEL
LIN {X 0,Y 453.503,Z 1030.234,A -85,B 0,C 180,E1 21895.463,E2 21895.463} C_VEL
LIN {X 0,Y 451.774,Z 1043.074,A -85,B 0,C 180,E1 21892.925,E2 21892.925} C_VEL
LIN {X 0,Y 450.319,Z 1055.465,A -85,B 0,C 180,E1 21890.084,E2 21890.084} C_VEL
LIN {X 0,Y 449.362,Z 1065.06,A -85,B 0,C 180,E1 21887.481,E2 21887.481} C_VEL
LIN {X 0,Y 448.615,Z 1074.346,A -85,B 0,C 180,E1 21884.455,E2 21884.455} C_VEL
LIN {X 0,Y 448.241,Z 1080.863,A -85,B 0,C 180,E1 21881.842,E2 21881.842} C_VEL
LIN {X 0,Y 448.022,Z 1086.635,A -85,B 0,C 180,E1 21878.858,E2 21878.858} C_VEL
LIN {X 0,Y 447.929,Z 1090.438,A -85,B 0,C 180,E1 21876.151,E2 21876.151} C_VEL
LIN {X 0,Y 447.886,Z 1092.985,A -85,B 0,C 180,E1 21873.199,E2 21873.199} C_VEL
LIN {X 0,Y 447.886,Z 1093.872,A -85,B 0,C 180,E1 21870.767,E2 21870.767} C_VEL
LIN {X 0,Y 447.91,Z 1093.595,A -85,B 0,C 180,E1 21867.953,E2 21867.953} C_VEL
LIN {X 0,Y 447.91,Z 1091.841,A -85,B 0,C 180,E1 21865.262,E2 21865.262} C_VEL
LIN {X 0,Y 447.954,Z 1088.68,A -85,B 0,C 180,E1 21862.433,E2 21862.433} C_VEL
LIN {X 0,Y 448.104,Z 1083.827,A -85,B 0,C 180,E1 21859.587,E2 21859.587} C_VEL
LIN {X 0,Y 448.435,Z 1077.516,A -85,B 0,C 180,E1 21856.723,E2 21856.723} C_VEL
LIN {X 0,Y 448.97,Z 1069.741,A -85,B 0,C 180,E1 21853.969,E2 21853.969} C_VEL
LIN {X 0,Y 449.823,Z 1060.441,A -85,B 0,C 180,E1 21851.198,E2 21851.198} C_VEL
LIN {X 0,Y 450.97,Z 1049.716,A -85,B 0,C 180,E1 21848.541,E2 21848.541} C_VEL
LIN {X 0,Y 452.561,Z 1037.096,A -85,B 0,C 180,E1 21845.846,E2 21845.846} C_VEL
LIN {X 0,Y 454.47,Z 1023.335,A -85,B 0,C 180,E1 21843.332,E2 21843.332} C_VEL
LIN {X 0,Y 456.824,Z 1007.519,A -85,B 0,C 180,E1 21840.843,E2 21840.843} C_VEL
LIN {X 0,Y 458.237,Z 996.793,A -85,B 0,C 180,E1 21839.442,E2 21839.442} C_VEL
LIN {X 0,Y 460.513,Z 978.615,A -85,B 0,C 180,E1 21837.396,E2 21837.396} C_VEL
LIN {X 0,Y 462.854,Z 959.321,A -85,B 0,C 180,E1 21835.53,E2 21835.53} C_VEL
LIN {X 0,Y 465.084,Z 940.126,A -85,B 0,C 180,E1 21833.909,E2 21833.909} C_VEL
LIN {X 0,Y 467.282,Z 919.288,A -85,B 0,C 180,E1 21832.423,E2 21832.423} C_VEL
LIN {X 0,Y 469.591,Z 896.349,A -85,B 0,C 180,E1 21831.035,E2 21831.035} C_VEL
LIN {X 0,Y 471.393,Z 875.899,A -85,B 0,C 180,E1 21830.007,E2 21830.007} C_VEL
LIN {X 0,Y 473.272,Z 851.246,A -85,B 0,C 180,E1 21829.011,E2 21829.011} C_VEL
LIN {X 0,Y 474.844,Z 827.515,A -85,B 0,C 180,E1 21828.272,E2 21828.272} C_VEL
LIN {X 0,Y 475.903,Z 803.556,A -85,B 0,C 180,E1 21827.751,E2 21827.751} C_VEL
LIN {X 0,Y 480.099,Z 631.009,A -85,B 0,C 180,E1 21824.722,E2 21824.722} C_VEL
LIN {X 0,Y 483.777,Z 493.343,A -85,B 0,C 180,E1 21822.24,E2 21822.24} C_VEL
LIN {X 0,Y 480.807,Z 465.421,A -85,B 0,C 180,E1 21821.302,E2 21821.302} C_VEL
LIN {X 0,Y 481.695,Z 451.595,A -85,B 0,C 180,E1 21820.44,E2 21820.44} C_VEL
LIN {X 0,Y 472.191,Z 432.449,A -85,B 0,C 180,E1 21817.884,E2 21817.884} C_VEL
LIN {X 0,Y 462.724,Z 415.083,A -85,B 0,C 180,E1 21815.235,E2 21815.235} C_VEL
LIN {X 0,Y 456.8,Z 405.032,A -85,B 0,C 180,E1 21813.493,E2 21813.493} C_VEL
LIN {X 0,Y 454.481,Z 400.933,A -85,B 0,C 180,E1 21812.765,E2 21812.765} C_VEL
LIN {X 0,Y 452.238,Z 397.07,A -85,B 0,C 180,E1 21812.047,E2 21812.047} C_VEL
LIN {X 0,Y 449.58,Z 392.97,A -85,B 0,C 180,E1 21811.21,E2 21811.21} C_VEL
LIN {X 0,Y 449.122,Z 391.414,A -85,B 0,C 180,E1 21810.902,E2 21810.902} C_VEL
LIN {X 0,Y 449.096,Z 391.07,A -85,B 0,C 180,E1 21809.62,E2 21809.62} C_VEL
LIN {X 0,Y 449.055,Z 391.066,A -85,B 0,C 180,E1 21806.158,E2 21806.158} C_VEL
LIN {X 0,Y 449.074,Z 391.11,A -85,B 0,C 180,E1 21802.482,E2 21802.482} C_VEL
LIN {X 0,Y 449.115,Z 391.055,A -85,B 0,C 180,E1 21798.883,E2 21798.883} C_VEL
LIN {X 0,Y 449.072,Z 391.094,A -85,B 0,C 180,E1 21795.364,E2 21795.364} C_VEL
LIN {X 0,Y 449.059,Z 391.067,A -85,B 0,C 180,E1 21791.69,E2 21791.69} C_VEL
LIN {X 0,Y 449.091,Z 391.09,A -85,B 0,C 180,E1 21788.063,E2 21788.063} C_VEL
LIN {X 0,Y 449.106,Z 391.091,A -85,B 0,C 180,E1 21784.469,E2 21784.469} C_VEL
LIN {X 0,Y 449.066,Z 391.099,A -85,B 0,C 180,E1 21780.893,E2 21780.893} C_VEL
LIN {X 0,Y 449.067,Z 391.101,A -85,B 0,C 180,E1 21777.192,E2 21777.192} C_VEL
LIN {X 0,Y 449.112,Z 391.096,A -85,B 0,C 180,E1 21773.608,E2 21773.608} C_VEL
LIN {X 0,Y 449.096,Z 391.102,A -85,B 0,C 180,E1 21769.999,E2 21769.999} C_VEL
LIN {X 0,Y 449.066,Z 391.109,A -85,B 0,C 180,E1 21766.48,E2 21766.48} C_VEL
LIN {X 0,Y 449.093,Z 391.105,A -85,B 0,C 180,E1 21762.909,E2 21762.909} C_VEL
LIN {X 0,Y 449.13,Z 391.1,A -85,B 0,C 180,E1 21759.231,E2 21759.231} C_VEL
LIN {X 0,Y 449.077,Z 391.108,A -85,B 0,C 180,E1 21755.676,E2 21755.676} C_VEL
LIN {X 0,Y 449.071,Z 391.097,A -85,B 0,C 180,E1 21751.979,E2 21751.979} C_VEL
LIN {X 0,Y 449.108,Z 391.066,A -85,B 0,C 180,E1 21748.453,E2 21748.453} C_VEL
LIN {X 0,Y 449.093,Z 391.066,A -85,B 0,C 180,E1 21744.941,E2 21744.941} C_VEL
LIN {X 0,Y 449.072,Z 391.112,A -85,B 0,C 180,E1 21741.399,E2 21741.399} C_VEL
LIN {X 0,Y 449.123,Z 391.365,A -85,B 0,C 180,E1 21739.75,E2 21739.75} C_VEL
LIN {X 0,Y 450.363,Z 394.528,A -85,B 0,C 180,E1 21739.085,E2 21739.085} C_VEL
LIN {X 0,Y 451.861,Z 396.665,A -85,B 0,C 180,E1 21738.576,E2 21738.576} C_VEL
LIN {X 0,Y 453.91,Z 400.515,A -85,B 0,C 180,E1 21737.79,E2 21737.79} C_VEL
LIN {X 0,Y 461.248,Z 414.96,A -85,B 0,C 180,E1 21735.034,E2 21735.034} C_VEL
LIN {X 0,Y 468.531,Z 430.327,A -85,B 0,C 180,E1 21732.404,E2 21732.404} C_VEL
LIN {X 0,Y 474.649,Z 444.563,A -85,B 0,C 180,E1 21730.215,E2 21730.215} C_VEL
LIN {X 0,Y 472.296,Z 470.009,A -85,B 0,C 180,E1 21728.152,E2 21728.152} C_VEL
LIN {X 0,Y 476.906,Z 498.069,A -85,B 0,C 180,E1 21727.101,E2 21727.101} C_VEL
LIN {X 0,Y 474.972,Z 605.891,A -85,B 0,C 180,E1 21725.411,E2 21725.411} C_VEL
LIN {X 0,Y 474.115,Z 613.603,A -85,B 0,C 180,E1 21725.37,E2 21725.37} C_VEL
LIN {X 0,Y 469.068,Z 634.196,A -85,B 0,C 180,E1 21725.555,E2 21725.555} C_VEL
LIN {X 0,Y 468.419,Z 640.813,A -85,B 0,C 180,E1 21725.511,E2 21725.511} C_VEL
LIN {X 0,Y 466.864,Z 742.127,A -85,B 0,C 180,E1 21723.918,E2 21723.918} C_VEL
LIN {X 0,Y 466.011,Z 762.216,A -85,B 0,C 180,E1 21723.383,E2 21723.383} C_VEL
LIN {X 0,Y 464.706,Z 781.601,A -85,B 0,C 180,E1 21722.651,E2 21722.651} C_VEL
LIN {X 0,Y 462.992,Z 800.416,A -85,B 0,C 180,E1 21721.719,E2 21721.719} C_VEL
LIN {X 0,Y 460.883,Z 818.599,A -85,B 0,C 180,E1 21720.58,E2 21720.58} C_VEL
LIN {X 0,Y 458.492,Z 835.854,A -85,B 0,C 180,E1 21719.242,E2 21719.242} C_VEL
LIN {X 0,Y 455.794,Z 852.954,A -85,B 0,C 180,E1 21717.636,E2 21717.636} C_VEL
LIN {X 0,Y 453.12,Z 868.674,A -85,B 0,C 180,E1 21715.851,E2 21715.851} C_VEL
LIN {X 0,Y 450.554,Z 882.687,A -85,B 0,C 180,E1 21713.961,E2 21713.961} C_VEL
LIN {X 0,Y 448.001,Z 896.284,A -85,B 0,C 180,E1 21711.746,E2 21711.746} C_VEL
LIN {X 0,Y 445.849,Z 907.62,A -85,B 0,C 180,E1 21709.521,E2 21709.521} C_VEL
LIN {X 0,Y 443.957,Z 918.15,A -85,B 0,C 180,E1 21707.025,E2 21707.025} C_VEL
LIN {X 0,Y 442.445,Z 927.644,A -85,B 0,C 180,E1 21704.26,E2 21704.26} C_VEL
LIN {X 0,Y 441.421,Z 935.205,A -85,B 0,C 180,E1 21701.498,E2 21701.498} C_VEL
LIN {X 0,Y 440.83,Z 940.993,A -85,B 0,C 180,E1 21698.741,E2 21698.741} C_VEL
LIN {X 0,Y 440.512,Z 945.16,A -85,B 0,C 180,E1 21695.993,E2 21695.993} C_VEL
LIN {X 0,Y 440.339,Z 947.809,A -85,B 0,C 180,E1 21693.124,E2 21693.124} C_VEL
LIN {X 0,Y 440.291,Z 948.76,A -85,B 0,C 180,E1 21690.39,E2 21690.39} C_VEL
LIN {X 0,Y 440.316,Z 948.227,A -85,B 0,C 180,E1 21687.632,E2 21687.632} C_VEL
LIN {X 0,Y 440.432,Z 946.096,A -85,B 0,C 180,E1 21684.79,E2 21684.79} C_VEL
LIN {X 0,Y 440.706,Z 942.485,A -85,B 0,C 180,E1 21682.045,E2 21682.045} C_VEL
LIN {X 0,Y 441.197,Z 937.278,A -85,B 0,C 180,E1 21679.29,E2 21679.29} C_VEL
LIN {X 0,Y 442.151,Z 929.926,A -85,B 0,C 180,E1 21676.398,E2 21676.398} C_VEL
LIN {X 0,Y 443.494,Z 920.979,A -85,B 0,C 180,E1 21673.631,E2 21673.631} C_VEL
LIN {X 0,Y 445.356,Z 910.435,A -85,B 0,C 180,E1 21671.002,E2 21671.002} C_VEL
LIN {X 0,Y 447.392,Z 899.394,A -85,B 0,C 180,E1 21668.74,E2 21668.74} C_VEL
LIN {X 0,Y 449.809,Z 886.595,A -85,B 0,C 180,E1 21666.553,E2 21666.553} C_VEL
LIN {X 0,Y 452.325,Z 873.021,A -85,B 0,C 180,E1 21664.606,E2 21664.606} C_VEL
LIN {X 0,Y 455.104,Z 857.407,A -85,B 0,C 180,E1 21662.737,E2 21662.737} C_VEL
LIN {X 0,Y 457.707,Z 841.198,A -85,B 0,C 180,E1 21661.133,E2 21661.133} C_VEL
LIN {X 0,Y 460.161,Z 824.058,A -85,B 0,C 180,E1 21659.728,E2 21659.728} C_VEL
LIN {X 0,Y 462.367,Z 806.041,A -85,B 0,C 180,E1 21658.517,E2 21658.517} C_VEL
LIN {X 0,Y 464.239,Z 787.761,A -85,B 0,C 180,E1 21657.532,E2 21657.532} C_VEL
LIN {X 0,Y 465.67,Z 768.621,A -85,B 0,C 180,E1 21656.743,E2 21656.743} C_VEL
LIN {X 0,Y 466.635,Z 748.527,A -85,B 0,C 180,E1 21656.139,E2 21656.139} C_VEL
LIN {X 0,Y 467.186,Z 724.021,A -85,B 0,C 180,E1 21655.677,E2 21655.677} C_VEL
LIN {X 0,Y 471.026,Z 499.268,A -85,B 0,C 180,E1 21652.164,E2 21652.164} C_VEL
LIN {X 0,Y 466.169,Z 468.992,A -85,B 0,C 180,E1 21650.978,E2 21650.978} C_VEL
LIN {X 0,Y 468.27,Z 448.075,A -85,B 0,C 180,E1 21649.232,E2 21649.232} C_VEL
LIN {X 0,Y 460.682,Z 430.762,A -85,B 0,C 180,E1 21646.462,E2 21646.462} C_VEL
LIN {X 0,Y 453.115,Z 415.053,A -85,B 0,C 180,E1 21643.632,E2 21643.632} C_VEL
LIN {X 0,Y 447.628,Z 404.823,A -85,B 0,C 180,E1 21641.558,E2 21641.558} C_VEL
LIN {X 0,Y 446.024,Z 401.524,A -85,B 0,C 180,E1 21640.888,E2 21640.888} C_VEL
LIN {X 0,Y 444.015,Z 397.926,A -85,B 0,C 180,E1 21640.094,E2 21640.094} C_VEL
LIN {X 0,Y 441.374,Z 393.204,A -85,B 0,C 180,E1 21639.012,E2 21639.012} C_VEL
LIN {X 0,Y 441.144,Z 392.124,A -85,B 0,C 180,E1 21638.64,E2 21638.64} C_VEL
LIN {X 0,Y 441.157,Z 392.052,A -85,B 0,C 180,E1 21634.989,E2 21634.989} C_VEL
LIN {X 0,Y 441.188,Z 392.046,A -85,B 0,C 180,E1 21631.307,E2 21631.307} C_VEL
LIN {X 0,Y 441.148,Z 392.091,A -85,B 0,C 180,E1 21627.687,E2 21627.687} C_VEL
LIN {X 0,Y 441.137,Z 392.098,A -85,B 0,C 180,E1 21624.017,E2 21624.017} C_VEL
LIN {X 0,Y 441.167,Z 392.097,A -85,B 0,C 180,E1 21620.428,E2 21620.428} C_VEL
LIN {X 0,Y 441.187,Z 392.093,A -85,B 0,C 180,E1 21616.728,E2 21616.728} C_VEL
LIN {X 0,Y 441.143,Z 392.096,A -85,B 0,C 180,E1 21613.1,E2 21613.1} C_VEL
LIN {X 0,Y 441.134,Z 392.098,A -85,B 0,C 180,E1 21609.393,E2 21609.393} C_VEL
LIN {X 0,Y 441.155,Z 392.098,A -85,B 0,C 180,E1 21605.724,E2 21605.724} C_VEL
LIN {X 0,Y 441.181,Z 392.089,A -85,B 0,C 180,E1 21602.078,E2 21602.078} C_VEL
LIN {X 0,Y 441.14,Z 392.093,A -85,B 0,C 180,E1 21598.442,E2 21598.442} C_VEL
LIN {X 0,Y 441.129,Z 392.096,A -85,B 0,C 180,E1 21594.799,E2 21594.799} C_VEL
LIN {X 0,Y 441.158,Z 392.089,A -85,B 0,C 180,E1 21591.181,E2 21591.181} C_VEL
LIN {X 0,Y 441.174,Z 392.035,A -85,B 0,C 180,E1 21587.434,E2 21587.434} C_VEL
LIN {X 0,Y 441.131,Z 392.096,A -85,B 0,C 180,E1 21583.948,E2 21583.948} C_VEL
LIN {X 0,Y 441.12,Z 392.043,A -85,B 0,C 180,E1 21580.163,E2 21580.163} C_VEL
LIN {X 0,Y 441.161,Z 392.081,A -85,B 0,C 180,E1 21576.622,E2 21576.622} C_VEL
LIN {X 0,Y 441.169,Z 392.063,A -85,B 0,C 180,E1 21572.901,E2 21572.901} C_VEL
LIN {X 0,Y 441.202,Z 392.237,A -85,B 0,C 180,E1 21570.544,E2 21570.544} C_VEL
LIN {X 0,Y 441.419,Z 393.348,A -85,B 0,C 180,E1 21570.261,E2 21570.261} C_VEL
LIN {X 0,Y 443.116,Z 396.426,A -85,B 0,C 180,E1 21569.64,E2 21569.64} C_VEL
LIN {X 0,Y 444.372,Z 397.946,A -85,B 0,C 180,E1 21569.263,E2 21569.263} C_VEL
LIN {X 0,Y 446.419,Z 401.677,A -85,B 0,C 180,E1 21568.544,E2 21568.544} C_VEL
LIN {X 0,Y 447.529,Z 403.512,A -85,B 0,C 180,E1 21568.18,E2 21568.18} C_VEL
LIN {X 0,Y 450.92,Z 409.284,A -85,B 0,C 180,E1 21567.095,E2 21567.095} C_VEL
LIN {X 0,Y 458.016,Z 421.458,A -85,B 0,C 180,E1 21564.949,E2 21564.949} C_VEL
LIN {X 0,Y 467.324,Z 438.907,A -85,B 0,C 180,E1 21562.273,E2 21562.273} C_VEL
LIN {X 0,Y 475.598,Z 455.751,A -85,B 0,C 180,E1 21559.981,E2 21559.981} C_VEL
LIN {X 0,Y 474.85,Z 467.061,A -85,B 0,C 180,E1 21559.309,E2 21559.309} C_VEL
LIN {X 0,Y 477.887,Z 496.892,A -85,B 0,C 180,E1 21558.329,E2 21558.329} C_VEL
LIN {X 0,Y 472.055,Z 696.047,A -85,B 0,C 180,E1 21554.707,E2 21554.707} C_VEL
LIN {X 0,Y 468.826,Z 812.189,A -85,B 0,C 180,E1 21552.602,E2 21552.602} C_VEL
LIN {X 0,Y 467.307,Z 836.806,A -85,B 0,C 180,E1 21551.954,E2 21551.954} C_VEL
LIN {X 0,Y 465.482,Z 861.591,A -85,B 0,C 180,E1 21551.067,E2 21551.067} C_VEL
LIN {X 0,Y 463.442,Z 884.882,A -85,B 0,C 180,E1 21550.014,E2 21550.014} C_VEL
LIN {X 0,Y 461.276,Z 906.742,A -85,B 0,C 180,E1 21548.788,E2 21548.788} C_VEL
LIN {X 0,Y 458.86,Z 929.238,A -85,B 0,C 180,E1 21547.284,E2 21547.284} C_VEL
LIN {X 0,Y 456.402,Z 950.033,A -85,B 0,C 180,E1 21545.644,E2 21545.644} C_VEL
LIN {X 0,Y 453.94,Z 970.152,A -85,B 0,C 180,E1 21543.78,E2 21543.78} C_VEL
LIN {X 0,Y 451.563,Z 988.647,A -85,B 0,C 180,E1 21541.802,E2 21541.802} C_VEL
LIN {X 0,Y 449.253,Z 1006.214,A -85,B 0,C 180,E1 21539.61,E2 21539.61} C_VEL
LIN {X 0,Y 447.122,Z 1022.389,A -85,B 0,C 180,E1 21537.286,E2 21537.286} C_VEL
LIN {X 0,Y 445.433,Z 1033.812,A -85,B 0,C 180,E1 21535.23,E2 21535.23} C_VEL
LIN {X 0,Y 443.624,Z 1046.841,A -85,B 0,C 180,E1 21532.529,E2 21532.529} C_VEL
LIN {X 0,Y 442.254,Z 1057.861,A -85,B 0,C 180,E1 21529.824,E2 21529.824} C_VEL
LIN {X 0,Y 441.249,Z 1067.715,A -85,B 0,C 180,E1 21526.996,E2 21526.996} C_VEL
LIN {X 0,Y 440.604,Z 1075.436,A -85,B 0,C 180,E1 21524.309,E2 21524.309} C_VEL
LIN {X 0,Y 440.199,Z 1082.301,A -85,B 0,C 180,E1 21521.397,E2 21521.397} C_VEL
LIN {X 0,Y 440.016,Z 1087.255,A -85,B 0,C 180,E1 21518.625,E2 21518.625} C_VEL
LIN {X 0,Y 439.916,Z 1091.046,A -85,B 0,C 180,E1 21515.739,E2 21515.739} C_VEL
LIN {X 0,Y 439.889,Z 1093.121,A -85,B 0,C 180,E1 21512.997,E2 21512.997} C_VEL
LIN {X 0,Y 439.891,Z 1093.939,A -85,B 0,C 180,E1 21510.391,E2 21510.391} C_VEL
LIN {X 0,Y 439.904,Z 1093.324,A -85,B 0,C 180,E1 21507.395,E2 21507.395} C_VEL
LIN {X 0,Y 439.919,Z 1091.5,A -85,B 0,C 180,E1 21504.784,E2 21504.784} C_VEL
LIN {X 0,Y 439.999,Z 1087.874,A -85,B 0,C 180,E1 21501.769,E2 21501.769} C_VEL
LIN {X 0,Y 440.16,Z 1083.318,A -85,B 0,C 180,E1 21499.132,E2 21499.132} C_VEL
LIN {X 0,Y 440.538,Z 1076.462,A -85,B 0,C 180,E1 21496.079,E2 21496.079} C_VEL
LIN {X 0,Y 441.134,Z 1068.931,A -85,B 0,C 180,E1 21493.406,E2 21493.406} C_VEL
LIN {X 0,Y 442.141,Z 1058.895,A -85,B 0,C 180,E1 21490.446,E2 21490.446} C_VEL
LIN {X 0,Y 443.395,Z 1048.568,A -85,B 0,C 180,E1 21487.877,E2 21487.877} C_VEL
LIN {X 0,Y 445.242,Z 1035.14,A -85,B 0,C 180,E1 21485.027,E2 21485.027} C_VEL
LIN {X 0,Y 446.892,Z 1024.016,A -85,B 0,C 180,E1 21482.987,E2 21482.987} C_VEL
